gfCNCPoint5[4835] = {X 411.3483, Y 48.2525, Z -6.3333, A 0.000, B 0.000, C 0.000 }
gfCNCPoint5[4836] = {X 410.5596, Y 48.7481, Z -6.3333, A 0.000, B 0.000, C 0.000 }
gfCNCPoint5[4837] = {X 409.6803, Y 49.0557, Z -6.3333, A 0.000, B 0.000, C 0.000 }
gfCNCPoint5[4838] = {X 408.7547, Y 49.1600, Z -6.3333, A 0.000, B 0.000, C 0.000 }
gfCNCPoint5[4839] = {X 402.3112, Y 49.1600, Z -6.3333, A 0.000, B 0.000, C 0.000 }
gfCNCPoint5[4840] = {X 401.3900, Y 49.0567, Z -6.3333, A 0.000, B 0.000, C 0.000 }
gfCNCPoint5[4841] = {X 400.5146, Y 48.7520, Z -6.3333, A 0.000, B 0.000, C 0.000 }
gfCNCPoint5[4842] = {X 399.7283, Y 48.2610, Z -6.3333, A 0.000, B 0.000, C 0.000 }
gfCNCPoint5[4843] = {X 399.0703, Y 47.6081, Z -6.3333, A 0.000, B 0.000, C 0.000 }
gfCNCPoint5[4844] = {X 398.5732, Y 46.8257, Z -6.3333, A 0.000, B 0.000, C 0.000 }
gfCNCPoint5[4845] = {X 398.2617, Y 45.9526, Z -6.3333, A 0.000, B 0.000, C 0.000 }
gfCNCPoint5[4846] = {X 398.1513, Y 45.0322, Z -6.3333, A 0.000, B 0.000, C 0.000 }
gfCNCPoint5[4847] = {X 398.1516, Y 44.1549, Z -6.3333, A 0.000, B 0.000, C 0.000 }
gfCNCPoint5[4848] = {X 398.2616, Y 43.2570, Z -6.3333, A 0.000, B 0.000, C 0.000 }
gfCNCPoint5[4849] = {X 398.5630, Y 42.4041, Z -6.3333, A 0.000, B 0.000, C 0.000 }
gfCNCPoint5[4850] = {X 399.0417, Y 41.6366, Z -6.3333, A 0.000, B 0.000, C 0.000 }
gfCNCPoint5[4851] = {X 399.6750, Y 40.9907, Z -6.3333, A 0.000, B 0.000, C 0.000 }
gfCNCPoint5[4852] = {X 399.6327, Y 31.5586, Z -6.3333, A 0.000, B 0.000, C 0.000 }
gfCNCPoint5[4853] = {X 393.6589, Y 21.1703, Z -6.3333, A 0.000, B 0.000, C 0.000 }
gfCNCPoint5[4854] = {X 392.7687, Y 19.6558, Z -6.3333, A 0.000, B 0.000, C 0.000 }
gfCNCPoint5[4855] = {X 391.8499, Y 18.1584, Z -6.3333, A 0.000, B 0.000, C 0.000 }
gfCNCPoint5[4856] = {X 391.3454, Y 17.4581, Z -6.3333, A 0.000, B 0.000, C 0.000 }
gfCNCPoint5[4857] = {X 390.7551, Y 16.8285, Z -6.3333, A 0.000, B 0.000, C 0.000 }
gfCNCPoint5[4858] = {X 389.9029, Y 16.3569, Z -6.3333, A 0.000, B 0.000, C 0.000 }
gfCNCPoint5[4859] = {X 389.1837, Y 15.7000, Z -6.3333, A 0.000, B 0.000, C 0.000 }
gfCNCPoint5[4860] = {X 388.6371, Y 14.8939, Z -6.3333, A 0.000, B 0.000, C 0.000 }
gfCNCPoint5[4861] = {X 388.2928, Y 13.9828, Z -6.3333, A 0.000, B 0.000, C 0.000 }
gfCNCPoint5[4862] = {X 388.1698, Y 13.0166, Z -6.3333, A 0.000, B 0.000, C 0.000 }
gfCNCPoint5[4863] = {X 388.1696, Y 12.1868, Z -6.3333, A 0.000, B 0.000, C 0.000 }
gfCNCPoint5[4864] = {X 388.2739, Y 11.2611, Z -6.3333, A 0.000, B 0.000, C 0.000 }
gfCNCPoint5[4865] = {X 388.5816, Y 10.3819, Z -6.3333, A 0.000, B 0.000, C 0.000 }
gfCNCPoint5[4866] = {X 389.0772, Y 9.5931, Z -6.3333, A 0.000, B 0.000, C 0.000 }
gfCNCPoint5[4867] = {X 389.7359, Y 8.9344, Z -6.3333, A 0.000, B 0.000, C 0.000 }
gfCNCPoint5[4868] = {X 390.5247, Y 8.4388, Z -6.3333, A 0.000, B 0.000, C 0.000 }
gfCNCPoint5[4869] = {X 391.4039, Y 8.1311, Z -6.3333, A 0.000, B 0.000, C 0.000 }
gfCNCPoint5[4870] = {X 392.3296, Y 8.0268, Z -6.3333, A 0.000, B 0.000, C 0.000 }
gfCNCPoint5[4871] = {X 399.1118, Y 8.0268, Z -6.3333, A 0.000, B 0.000, C 0.000 }
gfCNCPoint5[4872] = {X 400.0374, Y 8.1311, Z -6.3333, A 0.000, B 0.000, C 0.000 }
gfCNCPoint5[4873] = {X 400.9167, Y 8.4388, Z -6.3333, A 0.000, B 0.000, C 0.000 }
gfCNCPoint5[4874] = {X 401.7055, Y 8.9344, Z -6.3333, A 0.000, B 0.000, C 0.000 }
gfCNCPoint5[4875] = {X 402.3642, Y 9.5931, Z -6.3333, A 0.000, B 0.000, C 0.000 }
gfCNCPoint5[4876] = {X 402.8598, Y 10.3819, Z -6.3333, A 0.000, B 0.000, C 0.000 }
gfCNCPoint5[4877] = {X 403.1675, Y 11.2611, Z -6.3333, A 0.000, B 0.000, C 0.000 }
gfCNCPoint5[4878] = {X 403.2718, Y 12.1868, Z -6.3333, A 0.000, B 0.000, C 0.000 }
gfCNCPoint5[4879] = {X 403.2718, Y 12.9782, Z -6.3333, A 0.000, B 0.000, C 0.000 }
gfCNCPoint5[4880] = {X 403.1639, Y 13.9192, Z -6.3333, A 0.000, B 0.000, C 0.000 }
gfCNCPoint5[4881] = {X 402.8459, Y 14.8115, Z -6.3333, A 0.000, B 0.000, C 0.000 }
gfCNCPoint5[4882] = {X 405.3514, Y 19.1340, Z -6.3333, A 0.000, B 0.000, C 0.000 }
gfCNCPoint5[4883] = {X 408.0546, Y 14.7644, Z -6.3333, A 0.000, B 0.000, C 0.000 }
gfCNCPoint5[4884] = {X 407.7575, Y 13.9111, Z -6.3333, A 0.000, B 0.000, C 0.000 }
gfCNCPoint5[4885] = {X 407.6517, Y 13.0137, Z -6.3333, A 0.000, B 0.000, C 0.000 }
gfCNCPoint5[4886] = {X 407.6515, Y 12.1868, Z -6.3333, A 0.000, B 0.000, C 0.000 }
gfCNCPoint5[4887] = {X 407.7558, Y 11.2611, Z -6.3333, A 0.000, B 0.000, C 0.000 }
gfCNCPoint5[4888] = {X 408.0635, Y 10.3819, Z -6.3333, A 0.000, B 0.000, C 0.000 }
gfCNCPoint5[4889] = {X 408.5591, Y 9.5931, Z -6.3333, A 0.000, B 0.000, C 0.000 }
gfCNCPoint5[4890] = {X 409.2178, Y 8.9344, Z -6.3333, A 0.000, B 0.000, C 0.000 }
gfCNCPoint5[4891] = {X 410.0066, Y 8.4388, Z -6.3333, A 0.000, B 0.000, C 0.000 }
gfCNCPoint5[4892] = {X 410.8859, Y 8.1311, Z -6.3333, A 0.000, B 0.000, C 0.000 }
gfCNCPoint5[4893] = {X 411.8115, Y 8.0268, Z -6.3333, A 0.000, B 0.000, C 0.000 }
gfCNCPoint5[4894] = {X 419.3245, Y 8.0268, Z -6.3333, A 0.000, B 0.000, C 0.000 }
gfCNCPoint5[4895] = {X 420.2501, Y 8.1311, Z -6.3333, A 0.000, B 0.000, C 0.000 }
gfCNCPoint5[4896] = {X 421.1294, Y 8.4388, Z -6.3333, A 0.000, B 0.000, C 0.000 }
gfCNCPoint5[4897] = {X 421.9182, Y 8.9344, Z -6.3333, A 0.000, B 0.000, C 0.000 }
gfCNCPoint5[4898] = {X 422.5769, Y 9.5931, Z -6.3333, A 0.000, B 0.000, C 0.000 }
gfCNCPoint5[4899] = {X 423.0725, Y 10.3819, Z -6.3333, A 0.000, B 0.000, C 0.000 }
gfCNCPoint5[4900] = {X 423.3802, Y 11.2611, Z -6.3333, A 0.000, B 0.000, C 0.000 }
gfCNCPoint5[4901] = {X 423.4845, Y 12.1868, Z -6.3333, A 0.000, B 0.000, C 0.000 }
gfCNCPoint5[4902] = {X 423.4845, Y 12.9791, Z -6.3333, A 0.000, B 0.000, C 0.000 }
gfCNCPoint5[4903] = {X 423.3938, Y 13.8210, Z -6.3333, A 0.000, B 0.000, C 0.000 }
gfCNCPoint5[4904] = {X 423.1369, Y 14.6279, Z -6.3333, A 0.000, B 0.000, C 0.000 }
gfCNCPoint5[4905] = {X 422.7241, Y 15.3673, Z -6.3333, A 0.000, B 0.000, C 0.000 }
gfCNCPoint5[4906] = {X 422.1721, Y 16.0094, Z -6.3333, A 0.000, B 0.000, C 0.000 }
gfCNCPoint5[4907] = {X 421.5030, Y 16.5285, Z -6.3333, A 0.000, B 0.000, C 0.000 }
gfCNCPoint5[4908] = {X 420.7439, Y 16.9036, Z -6.3333, A 0.000, B 0.000, C 0.000 }
gfCNCPoint5[4909] = {X 420.0063, Y 17.8914, Z -6.3333, A 0.000, B 0.000, C 0.000 }
gfCNCPoint5[4910] = {X 419.3400, Y 18.9286, Z -6.3333, A 0.000, B 0.000, C 0.000 }
gfCNCPoint5[4911] = {X 417.8582, Y 21.3274, Z -6.3333, A 0.000, B 0.000, C 0.000 }
gfCNCPoint5[4912] = {X 416.0154, Y 24.2871, Z -6.3333, A 0.000, B 0.000, C 0.000 }
gfCNCPoint5[4913] = {X 419.4109, Y 26.4014, Z -6.3333, A 0.000, B 0.000, C 0.000 }
gfCNCPoint5[4914] = {X 415.9475, Y 24.2448, Z -6.3333, A 0.000, B 0.000, C 0.000 }
gfCNCPoint5[4915] = {X 411.3076, Y 31.6967, Z -6.3333, A 0.000, B 0.000, C 0.000 }
gfCNCPoint5[4916] = {X 411.3082, Y 41.0089, Z -6.3333, A 0.000, B 0.000, C 0.000 }
gfCNCPoint5[4917] = {X 411.9451, Y 41.6632, Z -6.3333, A 0.000, B 0.000, C 0.000 }
gfCNCPoint5[4918] = {X 412.4256, Y 42.4397, Z -6.3333, A 0.000, B 0.000, C 0.000 }
gfCNCPoint5[4919] = {X 412.7269, Y 43.3017, Z -6.3333, A 0.000, B 0.000, C 0.000 }
gfCNCPoint5[4920] = {X 412.8347, Y 44.2085, Z -6.3333, A 0.000, B 0.000, C 0.000 }
gfCNCPoint5[4921] = {X 412.8347, Y 45.0002, Z -6.3333, A 0.000, B 0.000, C 0.000 }
gfCNCPoint5[4922] = {X 412.7324, Y 45.9080, Z -6.3333, A 0.000, B 0.000, C 0.000 }
gfCNCPoint5[4923] = {X 412.4306, Y 46.7704, Z -6.3333, A 0.000, B 0.000, C 0.000 }
gfCNCPoint5[4924] = {X 411.9445, Y 47.5439, Z -6.3333, A 0.000, B 0.000, C 0.000 }
gfCNCPoint5[4925] = {X 411.2985, Y 48.1899, Z -6.3333, A 0.000, B 0.000, C 0.000 }
gfCNCPoint5[4926] = {X 410.5249, Y 48.6760, Z -6.3333, A 0.000, B 0.000, C 0.000 }
gfCNCPoint5[4927] = {X 409.6625, Y 48.9777, Z -6.3333, A 0.000, B 0.000, C 0.000 }
gfCNCPoint5[4928] = {X 408.7547, Y 49.0800, Z -6.3333, A 0.000, B 0.000, C 0.000 }
gfCNCPoint5[4929] = {X 402.3112, Y 49.0800, Z -6.3333, A 0.000, B 0.000, C 0.000 }
gfCNCPoint5[4930] = {X 401.4077, Y 48.9787, Z -6.3333, A 0.000, B 0.000, C 0.000 }
gfCNCPoint5[4931] = {X 400.5491, Y 48.6799, Z -6.3333, A 0.000, B 0.000, C 0.000 }
gfCNCPoint5[4932] = {X 399.7780, Y 48.1983, Z -6.3333, A 0.000, B 0.000, C 0.000 }
gfCNCPoint5[4933] = {X 399.1326, Y 47.5579, Z -6.3333, A 0.000, B 0.000, C 0.000 }
gfCNCPoint5[4934] = {X 398.6451, Y 46.7906, Z -6.3333, A 0.000, B 0.000, C 0.000 }
gfCNCPoint5[4935] = {X 398.3396, Y 45.9343, Z -6.3333, A 0.000, B 0.000, C 0.000 }
gfCNCPoint5[4936] = {X 398.2313, Y 45.0316, Z -6.3333, A 0.000, B 0.000, C 0.000 }
gfCNCPoint5[4937] = {X 398.2316, Y 44.1559, Z -6.3333, A 0.000, B 0.000, C 0.000 }
gfCNCPoint5[4938] = {X 398.3416, Y 43.2661, Z -6.3333, A 0.000, B 0.000, C 0.000 }
gfCNCPoint5[4939] = {X 398.6434, Y 42.4218, Z -6.3333, A 0.000, B 0.000, C 0.000 }
gfCNCPoint5[4940] = {X 399.1223, Y 41.6638, Z -6.3333, A 0.000, B 0.000, C 0.000 }
gfCNCPoint5[4941] = {X 399.7552, Y 41.0287, Z -6.3333, A 0.000, B 0.000, C 0.000 }
gfCNCPoint5[4942] = {X 399.7126, Y 31.5371, Z -6.3333, A 0.000, B 0.000, C 0.000 }
gfCNCPoint5[4943] = {X 393.7283, Y 21.1304, Z -6.3333, A 0.000, B 0.000, C 0.000 }
gfCNCPoint5[4944] = {X 392.8373, Y 19.6146, Z -6.3333, A 0.000, B 0.000, C 0.000 }
gfCNCPoint5[4945] = {X 391.9177, Y 18.1159, Z -6.3333, A 0.000, B 0.000, C 0.000 }
gfCNCPoint5[4946] = {X 391.4024, Y 17.4015, Z -6.3333, A 0.000, B 0.000, C 0.000 }
gfCNCPoint5[4947] = {X 390.7989, Y 16.7600, Z -6.3333, A 0.000, B 0.000, C 0.000 }
gfCNCPoint5[4948] = {X 389.9591, Y 16.2987, Z -6.3333, A 0.000, B 0.000, C 0.000 }
gfCNCPoint5[4949] = {X 389.2500, Y 15.6543, Z -6.3333, A 0.000, B 0.000, C 0.000 }
gfCNCPoint5[4950] = {X 388.7108, Y 14.8622, Z -6.3333, A 0.000, B 0.000, C 0.000 }
gfCNCPoint5[4951] = {X 388.3711, Y 13.9663, Z -6.3333, A 0.000, B 0.000, C 0.000 }
gfCNCPoint5[4952] = {X 388.2498, Y 13.0158, Z -6.3333, A 0.000, B 0.000, C 0.000 }
gfCNCPoint5[4953] = {X 388.2496, Y 12.1868, Z -6.3333, A 0.000, B 0.000, C 0.000 }
gfCNCPoint5[4954] = {X 388.3519, Y 11.2789, Z -6.3333, A 0.000, B 0.000, C 0.000 }
gfCNCPoint5[4955] = {X 388.6537, Y 10.4166, Z -6.3333, A 0.000, B 0.000, C 0.000 }
gfCNCPoint5[4956] = {X 389.1398, Y 9.6430, Z -6.3333, A 0.000, B 0.000, C 0.000 }
gfCNCPoint5[4957] = {X 389.7858, Y 8.9969, Z -6.3333, A 0.000, B 0.000, C 0.000 }
gfCNCPoint5[4958] = {X 390.5594, Y 8.5109, Z -6.3333, A 0.000, B 0.000, C 0.000 }
gfCNCPoint5[4959] = {X 391.4217, Y 8.2091, Z -6.3333, A 0.000, B 0.000, C 0.000 }
gfCNCPoint5[4960] = {X 392.3296, Y 8.1068, Z -6.3333, A 0.000, B 0.000, C 0.000 }
gfCNCPoint5[4961] = {X 399.1118, Y 8.1068, Z -6.3333, A 0.000, B 0.000, C 0.000 }
gfCNCPoint5[4962] = {X 400.0196, Y 8.2091, Z -6.3333, A 0.000, B 0.000, C 0.000 }
gfCNCPoint5[4963] = {X 400.8820, Y 8.5109, Z -6.3333, A 0.000, B 0.000, C 0.000 }
gfCNCPoint5[4964] = {X 401.6556, Y 8.9969, Z -6.3333, A 0.000, B 0.000, C 0.000 }
gfCNCPoint5[4965] = {X 402.3016, Y 9.6430, Z -6.3333, A 0.000, B 0.000, C 0.000 }
gfCNCPoint5[4966] = {X 402.7877, Y 10.4166, Z -6.3333, A 0.000, B 0.000, C 0.000 }
gfCNCPoint5[4967] = {X 403.0895, Y 11.2789, Z -6.3333, A 0.000, B 0.000, C 0.000 }
gfCNCPoint5[4968] = {X 403.1918, Y 12.1868, Z -6.3333, A 0.000, B 0.000, C 0.000 }
gfCNCPoint5[4969] = {X 403.1918, Y 12.9782, Z -6.3333, A 0.000, B 0.000, C 0.000 }
gfCNCPoint5[4970] = {X 403.0811, Y 13.9219, Z -6.3333, A 0.000, B 0.000, C 0.000 }
gfCNCPoint5[4971] = {X 402.7551, Y 14.8144, Z -6.3333, A 0.000, B 0.000, C 0.000 }
gfCNCPoint5[4972] = {X 405.3492, Y 19.2896, Z -6.3333, A 0.000, B 0.000, C 0.000 }
gfCNCPoint5[4973] = {X 408.1457, Y 14.7691, Z -6.3333, A 0.000, B 0.000, C 0.000 }
gfCNCPoint5[4974] = {X 408.1090, Y 14.6919, Z -6.3333, A 0.000, B 0.000, C 0.000 }
gfCNCPoint5[4975] = {X 408.0738, Y 14.6138, Z -6.3333, A 0.000, B 0.000, C 0.000 }
gfCNCPoint5[4976] = {X 407.8217, Y 13.8308, Z -6.3333, A 0.000, B 0.000, C 0.000 }
gfCNCPoint5[4977] = {X 407.7317, Y 13.0131, Z -6.3333, A 0.000, B 0.000, C 0.000 }
gfCNCPoint5[4978] = {X 407.7315, Y 12.1868, Z -6.3333, A 0.000, B 0.000, C 0.000 }
gfCNCPoint5[4979] = {X 407.8338, Y 11.2789, Z -6.3333, A 0.000, B 0.000, C 0.000 }
gfCNCPoint5[4980] = {X 408.1356, Y 10.4166, Z -6.3333, A 0.000, B 0.000, C 0.000 }
gfCNCPoint5[4981] = {X 408.6217, Y 9.6430, Z -6.3333, A 0.000, B 0.000, C 0.000 }
gfCNCPoint5[4982] = {X 409.2677, Y 8.9969, Z -6.3333, A 0.000, B 0.000, C 0.000 }
gfCNCPoint5[4983] = {X 410.0413, Y 8.5109, Z -6.3333, A 0.000, B 0.000, C 0.000 }
gfCNCPoint5[4984] = {X 410.9037, Y 8.2091, Z -6.3333, A 0.000, B 0.000, C 0.000 }
gfCNCPoint5[4985] = {X 411.8115, Y 8.1068, Z -6.3333, A 0.000, B 0.000, C 0.000 }
gfCNCPoint5[4986] = {X 419.3245, Y 8.1068, Z -6.3333, A 0.000, B 0.000, C 0.000 }
gfCNCPoint5[4987] = {X 420.2323, Y 8.2091, Z -6.3333, A 0.000, B 0.000, C 0.000 }
gfCNCPoint5[4988] = {X 421.0947, Y 8.5109, Z -6.3333, A 0.000, B 0.000, C 0.000 }
gfCNCPoint5[4989] = {X 421.8683, Y 8.9969, Z -6.3333, A 0.000, B 0.000, C 0.000 }
gfCNCPoint5[4990] = {X 422.5143, Y 9.6430, Z -6.3333, A 0.000, B 0.000, C 0.000 }
gfCNCPoint5[4991] = {X 423.0004, Y 10.4166, Z -6.3333, A 0.000, B 0.000, C 0.000 }
gfCNCPoint5[4992] = {X 423.3022, Y 11.2789, Z -6.3333, A 0.000, B 0.000, C 0.000 }
gfCNCPoint5[4993] = {X 423.4045, Y 12.1868, Z -6.3333, A 0.000, B 0.000, C 0.000 }
gfCNCPoint5[4994] = {X 423.4045, Y 12.9785, Z -6.3333, A 0.000, B 0.000, C 0.000 }
gfCNCPoint5[4995] = {X 423.3147, Y 13.8081, Z -6.3333, A 0.000, B 0.000, C 0.000 }
gfCNCPoint5[4996] = {X 423.0606, Y 14.6028, Z -6.3333, A 0.000, B 0.000, C 0.000 }
gfCNCPoint5[4997] = {X 422.6523, Y 15.3304, Z -6.3333, A 0.000, B 0.000, C 0.000 }
gfCNCPoint5[4998] = {X 422.1064, Y 15.9614, Z -6.3333, A 0.000, B 0.000, C 0.000 }
gfCNCPoint5[4999] = {X 421.4452, Y 16.4703, Z -6.3333, A 0.000, B 0.000, C 0.000 }
gfCNCPoint5[5000] = {X 420.6953, Y 16.8362, Z -6.3333, A 0.000, B 0.000, C 0.000 }
gfCNCPoint5[5001] = {X 419.9471, Y 17.8364, Z -6.3333, A 0.000, B 0.000, C 0.000 }
gfCNCPoint5[5002] = {X 419.2716, Y 18.8871, Z -6.3333, A 0.000, B 0.000, C 0.000 }
gfCNCPoint5[5003] = {X 417.7903, Y 21.2852, Z -6.3333, A 0.000, B 0.000, C 0.000 }
gfCNCPoint5[5004] = {X 415.9475, Y 24.2448, Z -6.3333, A 0.000, B 0.000, C 0.000 }
gfCNCPoint5[5005] = {X 419.3430, Y 26.3591, Z -6.3333, A 0.000, B 0.000, C 0.000 }
gfCNCPoint5[5006] = {X 415.8795, Y 24.2025, Z -6.3333, A 0.000, B 0.000, C 0.000 }
gfCNCPoint5[5007] = {X 411.2276, Y 31.6738, Z -6.3333, A 0.000, B 0.000, C 0.000 }
gfCNCPoint5[5008] = {X 411.2282, Y 41.0468, Z -6.3333, A 0.000, B 0.000, C 0.000 }
gfCNCPoint5[5009] = {X 411.8646, Y 41.6902, Z -6.3333, A 0.000, B 0.000, C 0.000 }
gfCNCPoint5[5010] = {X 412.3452, Y 42.4571, Z -6.3333, A 0.000, B 0.000, C 0.000 }
gfCNCPoint5[5011] = {X 412.6467, Y 43.3103, Z -6.3333, A 0.000, B 0.000, C 0.000 }
gfCNCPoint5[5012] = {X 412.7547, Y 44.2089, Z -6.3333, A 0.000, B 0.000, C 0.000 }
gfCNCPoint5[5013] = {X 412.7545, Y 45.0384, Z -6.3333, A 0.000, B 0.000, C 0.000 }
gfCNCPoint5[5014] = {X 412.6469, Y 45.9222, Z -6.3333, A 0.000, B 0.000, C 0.000 }
gfCNCPoint5[5015] = {X 412.3466, Y 46.7602, Z -6.3333, A 0.000, B 0.000, C 0.000 }
gfCNCPoint5[5016] = {X 411.8683, Y 47.5111, Z -6.3333, A 0.000, B 0.000, C 0.000 }
gfCNCPoint5[5017] = {X 411.2357, Y 48.1376, Z -6.3333, A 0.000, B 0.000, C 0.000 }
gfCNCPoint5[5018] = {X 410.4803, Y 48.6086, Z -6.3333, A 0.000, B 0.000, C 0.000 }
gfCNCPoint5[5019] = {X 409.6394, Y 48.9009, Z -6.3333, A 0.000, B 0.000, C 0.000 }
gfCNCPoint5[5020] = {X 408.7547, Y 49.0000, Z -6.3333, A 0.000, B 0.000, C 0.000 }
gfCNCPoint5[5021] = {X 402.3112, Y 49.0000, Z -6.3333, A 0.000, B 0.000, C 0.000 }
gfCNCPoint5[5022] = {X 401.4211, Y 48.8997, Z -6.3333, A 0.000, B 0.000, C 0.000 }
gfCNCPoint5[5023] = {X 400.5757, Y 48.6039, Z -6.3333, A 0.000, B 0.000, C 0.000 }
gfCNCPoint5[5024] = {X 399.8172, Y 48.1273, Z -6.3333, A 0.000, B 0.000, C 0.000 }
gfCNCPoint5[5025] = {X 399.1839, Y 47.4939, Z -6.3333, A 0.000, B 0.000, C 0.000 }
gfCNCPoint5[5026] = {X 398.7073, Y 46.7355, Z -6.3333, A 0.000, B 0.000, C 0.000 }
gfCNCPoint5[5027] = {X 398.4115, Y 45.8901, Z -6.3333, A 0.000, B 0.000, C 0.000 }
gfCNCPoint5[5028] = {X 398.3112, Y 45.0000, Z -6.3333, A 0.000, B 0.000, C 0.000 }
gfCNCPoint5[5029] = {X 398.3115, Y 44.1569, Z -6.3333, A 0.000, B 0.000, C 0.000 }
gfCNCPoint5[5030] = {X 398.4217, Y 43.2753, Z -6.3333, A 0.000, B 0.000, C 0.000 }
gfCNCPoint5[5031] = {X 398.7237, Y 42.4397, Z -6.3333, A 0.000, B 0.000, C 0.000 }
gfCNCPoint5[5032] = {X 399.2028, Y 41.6913, Z -6.3333, A 0.000, B 0.000, C 0.000 }
gfCNCPoint5[5033] = {X 399.8352, Y 41.0672, Z -6.3333, A 0.000, B 0.000, C 0.000 }
gfCNCPoint5[5034] = {X 399.8367, Y 31.5924, Z -6.3333, A 0.000, B 0.000, C 0.000 }
gfCNCPoint5[5035] = {X 393.7976, Y 21.0906, Z -6.3333, A 0.000, B 0.000, C 0.000 }
gfCNCPoint5[5036] = {X 392.9059, Y 19.5734, Z -6.3333, A 0.000, B 0.000, C 0.000 }
gfCNCPoint5[5037] = {X 391.9855, Y 18.0734, Z -6.3333, A 0.000, B 0.000, C 0.000 }
gfCNCPoint5[5038] = {X 391.4594, Y 17.3449, Z -6.3333, A 0.000, B 0.000, C 0.000 }
gfCNCPoint5[5039] = {X 390.8426, Y 16.6913, Z -6.3333, A 0.000, B 0.000, C 0.000 }
gfCNCPoint5[5040] = {X 390.0091, Y 16.2361, Z -6.3333, A 0.000, B 0.000, C 0.000 }
gfCNCPoint5[5041] = {X 389.3064, Y 15.5972, Z -6.3333, A 0.000, B 0.000, C 0.000 }
gfCNCPoint5[5042] = {X 388.7742, Y 14.8107, Z -6.3333, A 0.000, B 0.000, C 0.000 }
gfCNCPoint5[5043] = {X 388.4423, Y 13.9209, Z -6.3333, A 0.000, B 0.000, C 0.000 }
gfCNCPoint5[5044] = {X 388.3296, Y 12.9780, Z -6.3333, A 0.000, B 0.000, C 0.000 }
gfCNCPoint5[5045] = {X 388.3296, Y 12.1868, Z -6.3333, A 0.000, B 0.000, C 0.000 }
gfCNCPoint5[5046] = {X 388.4299, Y 11.2967, Z -6.3333, A 0.000, B 0.000, C 0.000 }
gfCNCPoint5[5047] = {X 388.7258, Y 10.4513, Z -6.3333, A 0.000, B 0.000, C 0.000 }
gfCNCPoint5[5048] = {X 389.2023, Y 9.6929, Z -6.3333, A 0.000, B 0.000, C 0.000 }
gfCNCPoint5[5049] = {X 389.8357, Y 9.0595, Z -6.3333, A 0.000, B 0.000, C 0.000 }
gfCNCPoint5[5050] = {X 390.5941, Y 8.5829, Z -6.3333, A 0.000, B 0.000, C 0.000 }
gfCNCPoint5[5051] = {X 391.4395, Y 8.2871, Z -6.3333, A 0.000, B 0.000, C 0.000 }
gfCNCPoint5[5052] = {X 392.3296, Y 8.1868, Z -6.3333, A 0.000, B 0.000, C 0.000 }
gfCNCPoint5[5053] = {X 399.1118, Y 8.1868, Z -6.3333, A 0.000, B 0.000, C 0.000 }
gfCNCPoint5[5054] = {X 400.0018, Y 8.2871, Z -6.3333, A 0.000, B 0.000, C 0.000 }
gfCNCPoint5[5055] = {X 400.8473, Y 8.5829, Z -6.3333, A 0.000, B 0.000, C 0.000 }
gfCNCPoint5[5056] = {X 401.6057, Y 9.0595, Z -6.3333, A 0.000, B 0.000, C 0.000 }
gfCNCPoint5[5057] = {X 402.2391, Y 9.6929, Z -6.3333, A 0.000, B 0.000, C 0.000 }
gfCNCPoint5[5058] = {X 402.7156, Y 10.4513, Z -6.3333, A 0.000, B 0.000, C 0.000 }
gfCNCPoint5[5059] = {X 403.0115, Y 11.2967, Z -6.3333, A 0.000, B 0.000, C 0.000 }
gfCNCPoint5[5060] = {X 403.1118, Y 12.1868, Z -6.3333, A 0.000, B 0.000, C 0.000 }
gfCNCPoint5[5061] = {X 403.1115, Y 13.0192, Z -6.3333, A 0.000, B 0.000, C 0.000 }
gfCNCPoint5[5062] = {X 402.9933, Y 13.9442, Z -6.3333, A 0.000, B 0.000, C 0.000 }
gfCNCPoint5[5063] = {X 402.6641, Y 14.8167, Z -6.3333, A 0.000, B 0.000, C 0.000 }
gfCNCPoint5[5064] = {X 405.2576, Y 19.3199, Z -6.3333, A 0.000, B 0.000, C 0.000 }
gfCNCPoint5[5065] = {X 405.3705, Y 19.4073, Z -6.3333, A 0.000, B 0.000, C 0.000 }
gfCNCPoint5[5066] = {X 408.1939, Y 14.8342, Z -6.3333, A 0.000, B 0.000, C 0.000 }
gfCNCPoint5[5067] = {X 408.2428, Y 14.7847, Z -6.3333, A 0.000, B 0.000, C 0.000 }
gfCNCPoint5[5068] = {X 408.1935, Y 14.6839, Z -6.3333, A 0.000, B 0.000, C 0.000 }
gfCNCPoint5[5069] = {X 408.1471, Y 14.5818, Z -6.3333, A 0.000, B 0.000, C 0.000 }
gfCNCPoint5[5070] = {X 407.8963, Y 13.7972, Z -6.3333, A 0.000, B 0.000, C 0.000 }
gfCNCPoint5[5071] = {X 407.8115, Y 12.9780, Z -6.3333, A 0.000, B 0.000, C 0.000 }
gfCNCPoint5[5072] = {X 407.8115, Y 12.1868, Z -6.3333, A 0.000, B 0.000, C 0.000 }
gfCNCPoint5[5073] = {X 407.9118, Y 11.2967, Z -6.3333, A 0.000, B 0.000, C 0.000 }
gfCNCPoint5[5074] = {X 408.2077, Y 10.4513, Z -6.3333, A 0.000, B 0.000, C 0.000 }
gfCNCPoint5[5075] = {X 408.6842, Y 9.6929, Z -6.3333, A 0.000, B 0.000, C 0.000 }
gfCNCPoint5[5076] = {X 409.3176, Y 9.0595, Z -6.3333, A 0.000, B 0.000, C 0.000 }
gfCNCPoint5[5077] = {X 410.0760, Y 8.5829, Z -6.3333, A 0.000, B 0.000, C 0.000 }
gfCNCPoint5[5078] = {X 410.9215, Y 8.2871, Z -6.3333, A 0.000, B 0.000, C 0.000 }
gfCNCPoint5[5079] = {X 411.8115, Y 8.1868, Z -6.3333, A 0.000, B 0.000, C 0.000 }
gfCNCPoint5[5080] = {X 419.3245, Y 8.1868, Z -6.3333, A 0.000, B 0.000, C 0.000 }
gfCNCPoint5[5081] = {X 420.2145, Y 8.2871, Z -6.3333, A 0.000, B 0.000, C 0.000 }
gfCNCPoint5[5082] = {X 421.0600, Y 8.5829, Z -6.3333, A 0.000, B 0.000, C 0.000 }
gfCNCPoint5[5083] = {X 421.8184, Y 9.0595, Z -6.3333, A 0.000, B 0.000, C 0.000 }
gfCNCPoint5[5084] = {X 422.4518, Y 9.6929, Z -6.3333, A 0.000, B 0.000, C 0.000 }
gfCNCPoint5[5085] = {X 422.9283, Y 10.4513, Z -6.3333, A 0.000, B 0.000, C 0.000 }
gfCNCPoint5[5086] = {X 423.2242, Y 11.2967, Z -6.3333, A 0.000, B 0.000, C 0.000 }
gfCNCPoint5[5087] = {X 423.3245, Y 12.1868, Z -6.3333, A 0.000, B 0.000, C 0.000 }
gfCNCPoint5[5088] = {X 423.3245, Y 12.9780, Z -6.3333, A 0.000, B 0.000, C 0.000 }
gfCNCPoint5[5089] = {X 423.2357, Y 13.7951, Z -6.3333, A 0.000, B 0.000, C 0.000 }
gfCNCPoint5[5090] = {X 422.9843, Y 14.5776, Z -6.3333, A 0.000, B 0.000, C 0.000 }
gfCNCPoint5[5091] = {X 422.5805, Y 15.2934, Z -6.3333, A 0.000, B 0.000, C 0.000 }
gfCNCPoint5[5092] = {X 422.0408, Y 15.9133, Z -6.3333, A 0.000, B 0.000, C 0.000 }
gfCNCPoint5[5093] = {X 421.3874, Y 16.4119, Z -6.3333, A 0.000, B 0.000, C 0.000 }
gfCNCPoint5[5094] = {X 420.6470, Y 16.7687, Z -6.3333, A 0.000, B 0.000, C 0.000 }
gfCNCPoint5[5095] = {X 419.8879, Y 17.7814, Z -6.3333, A 0.000, B 0.000, C 0.000 }
gfCNCPoint5[5096] = {X 419.2032, Y 18.8457, Z -6.3333, A 0.000, B 0.000, C 0.000 }
gfCNCPoint5[5097] = {X 417.7223, Y 21.2430, Z -6.3333, A 0.000, B 0.000, C 0.000 }
gfCNCPoint5[5098] = {X 415.8795, Y 24.2025, Z -6.3333, A 0.000, B 0.000, C 0.000 }
gfCNCPoint5[5099] = {X 419.3430, Y 26.3591, Z -6.3333, A 0.000, B 0.000, C 0.000 }
gfCNCPoint5[5100] = {X 419.3430, Y 26.3591, Z -3.3333, A 0.000, B 0.000, C 0.000 }
gfCNCPoint5[5101] = {X 419.3430, Y 26.3591, Z 11.0000, A 0.000, B 0.000, C 0.000 }
gfCNCPoint5[5102] = {X 352.3460, Y -3.5307, Z 11.0000, A 0.000, B 0.000, C 0.000 }
gfCNCPoint5[5103] = {X 352.3460, Y -3.5307, Z -3.3333, A 0.000, B 0.000, C 0.000 }
gfCNCPoint5[5104] = {X 352.3460, Y -3.5307, Z -6.3333, A 0.000, B 0.000, C 0.000 }
gfCNCPoint5[5105] = {X 351.5945, Y 0.4795, Z -6.3333, A 0.000, B 0.000, C 0.000 }
gfCNCPoint5[5106] = {X 351.8708, Y 0.5313, Z -6.3333, A 0.000, B 0.000, C 0.000 }
gfCNCPoint5[5107] = {X 353.8214, Y 1.0218, Z -6.3333, A 0.000, B 0.000, C 0.000 }
gfCNCPoint5[5108] = {X 355.7161, Y 1.6965, Z -6.3333, A 0.000, B 0.000, C 0.000 }
gfCNCPoint5[5109] = {X 357.5377, Y 2.5493, Z -6.3333, A 0.000, B 0.000, C 0.000 }
gfCNCPoint5[5110] = {X 359.2694, Y 3.5724, Z -6.3333, A 0.000, B 0.000, C 0.000 }
gfCNCPoint5[5111] = {X 360.8953, Y 4.7563, Z -6.3333, A 0.000, B 0.000, C 0.000 }
gfCNCPoint5[5112] = {X 362.4006, Y 6.0902, Z -6.3333, A 0.000, B 0.000, C 0.000 }
gfCNCPoint5[5113] = {X 363.7715, Y 7.5620, Z -6.3333, A 0.000, B 0.000, C 0.000 }
gfCNCPoint5[5114] = {X 365.1227, Y 9.3183, Z -6.3333, A 0.000, B 0.000, C 0.000 }
gfCNCPoint5[5115] = {X 366.3137, Y 11.1869, Z -6.3333, A 0.000, B 0.000, C 0.000 }
gfCNCPoint5[5116] = {X 367.3352, Y 13.1533, Z -6.3333, A 0.000, B 0.000, C 0.000 }
gfCNCPoint5[5117] = {X 368.1794, Y 15.2022, Z -6.3333, A 0.000, B 0.000, C 0.000 }
gfCNCPoint5[5118] = {X 368.8395, Y 17.3175, Z -6.3333, A 0.000, B 0.000, C 0.000 }
gfCNCPoint5[5119] = {X 369.3106, Y 19.4827, Z -6.3333, A 0.000, B 0.000, C 0.000 }
gfCNCPoint5[5120] = {X 369.6416, Y 21.8511, Z -6.3333, A 0.000, B 0.000, C 0.000 }
gfCNCPoint5[5121] = {X 369.7933, Y 24.2377, Z -6.3333, A 0.000, B 0.000, C 0.000 }
gfCNCPoint5[5122] = {X 369.7650, Y 26.6289, Z -6.3333, A 0.000, B 0.000, C 0.000 }
gfCNCPoint5[5123] = {X 369.5567, Y 29.0112, Z -6.3333, A 0.000, B 0.000, C 0.000 }
gfCNCPoint5[5124] = {X 369.1697, Y 31.3710, Z -6.3333, A 0.000, B 0.000, C 0.000 }
gfCNCPoint5[5125] = {X 368.6457, Y 33.4753, Z -6.3333, A 0.000, B 0.000, C 0.000 }
gfCNCPoint5[5126] = {X 367.9378, Y 35.5251, Z -6.3333, A 0.000, B 0.000, C 0.000 }
gfCNCPoint5[5127] = {X 367.0518, Y 37.5043, Z -6.3333, A 0.000, B 0.000, C 0.000 }
gfCNCPoint5[5128] = {X 365.9944, Y 39.3976, Z -6.3333, A 0.000, B 0.000, C 0.000 }
gfCNCPoint5[5129] = {X 364.7739, Y 41.1901, Z -6.3333, A 0.000, B 0.000, C 0.000 }
gfCNCPoint5[5130] = {X 364.6580, Y 41.3487, Z -6.3333, A 0.000, B 0.000, C 0.000 }
gfCNCPoint5[5131] = {X 363.2575, Y 43.0257, Z -6.3333, A 0.000, B 0.000, C 0.000 }
gfCNCPoint5[5132] = {X 361.6976, Y 44.5554, Z -6.3333, A 0.000, B 0.000, C 0.000 }
gfCNCPoint5[5133] = {X 359.9935, Y 45.9227, Z -6.3333, A 0.000, B 0.000, C 0.000 }
gfCNCPoint5[5134] = {X 358.1622, Y 47.1141, Z -6.3333, A 0.000, B 0.000, C 0.000 }
gfCNCPoint5[5135] = {X 356.2216, Y 48.1178, Z -6.3333, A 0.000, B 0.000, C 0.000 }
gfCNCPoint5[5136] = {X 354.0239, Y 48.9381, Z -6.3333, A 0.000, B 0.000, C 0.000 }
gfCNCPoint5[5137] = {X 351.7542, Y 49.5305, Z -6.3333, A 0.000, B 0.000, C 0.000 }
gfCNCPoint5[5138] = {X 349.4359, Y 49.8889, Z -6.3333, A 0.000, B 0.000, C 0.000 }
gfCNCPoint5[5139] = {X 347.0933, Y 50.0096, Z -6.3333, A 0.000, B 0.000, C 0.000 }
gfCNCPoint5[5140] = {X 345.0267, Y 49.9747, Z -6.3333, A 0.000, B 0.000, C 0.000 }
gfCNCPoint5[5141] = {X 342.9709, Y 49.7607, Z -6.3333, A 0.000, B 0.000, C 0.000 }
gfCNCPoint5[5142] = {X 340.9414, Y 49.3693, Z -6.3333, A 0.000, B 0.000, C 0.000 }
gfCNCPoint5[5143] = {X 338.9535, Y 48.8033, Z -6.3333, A 0.000, B 0.000, C 0.000 }
gfCNCPoint5[5144] = {X 337.0222, Y 48.0670, Z -6.3333, A 0.000, B 0.000, C 0.000 }
gfCNCPoint5[5145] = {X 335.1620, Y 47.1660, Z -6.3333, A 0.000, B 0.000, C 0.000 }
gfCNCPoint5[5146] = {X 333.5782, Y 46.1877, Z -6.3333, A 0.000, B 0.000, C 0.000 }
gfCNCPoint5[5147] = {X 332.0753, Y 45.0892, Z -6.3333, A 0.000, B 0.000, C 0.000 }
gfCNCPoint5[5148] = {X 330.6625, Y 43.8770, Z -6.3333, A 0.000, B 0.000, C 0.000 }
gfCNCPoint5[5149] = {X 329.7214, Y 43.8765, Z -6.3333, A 0.000, B 0.000, C 0.000 }
gfCNCPoint5[5150] = {X 328.8027, Y 43.6722, Z -6.3333, A 0.000, B 0.000, C 0.000 }
gfCNCPoint5[5151] = {X 327.9501, Y 43.2738, Z -6.3333, A 0.000, B 0.000, C 0.000 }
gfCNCPoint5[5152] = {X 327.2040, Y 42.7002, Z -6.3333, A 0.000, B 0.000, C 0.000 }
gfCNCPoint5[5153] = {X 326.5808, Y 42.0925, Z -6.3333, A 0.000, B 0.000, C 0.000 }
gfCNCPoint5[5154] = {X 325.9523, Y 41.3190, Z -6.3333, A 0.000, B 0.000, C 0.000 }
gfCNCPoint5[5155] = {X 325.5179, Y 40.4220, Z -6.3333, A 0.000, B 0.000, C 0.000 }
gfCNCPoint5[5156] = {X 325.3006, Y 39.4493, Z -6.3333, A 0.000, B 0.000, C 0.000 }
gfCNCPoint5[5157] = {X 325.3120, Y 38.4527, Z -6.3333, A 0.000, B 0.000, C 0.000 }
gfCNCPoint5[5158] = {X 325.5514, Y 37.4852, Z -6.3333, A 0.000, B 0.000, C 0.000 }
gfCNCPoint5[5159] = {X 326.0062, Y 36.5984, Z -6.3333, A 0.000, B 0.000, C 0.000 }
gfCNCPoint5[5160] = {X 330.2396, Y 30.2687, Z -6.3333, A 0.000, B 0.000, C 0.000 }
gfCNCPoint5[5161] = {X 330.8409, Y 29.5518, Z -6.3333, A 0.000, B 0.000, C 0.000 }
gfCNCPoint5[5162] = {X 331.5826, Y 28.9812, Z -6.3333, A 0.000, B 0.000, C 0.000 }
gfCNCPoint5[5163] = {X 332.4297, Y 28.5837, Z -6.3333, A 0.000, B 0.000, C 0.000 }
gfCNCPoint5[5164] = {X 333.3425, Y 28.3780, Z -6.3333, A 0.000, B 0.000, C 0.000 }
gfCNCPoint5[5165] = {X 334.2782, Y 28.3736, Z -6.3333, A 0.000, B 0.000, C 0.000 }
gfCNCPoint5[5166] = {X 335.1929, Y 28.5708, Z -6.3333, A 0.000, B 0.000, C 0.000 }
gfCNCPoint5[5167] = {X 336.0437, Y 28.9604, Z -6.3333, A 0.000, B 0.000, C 0.000 }
gfCNCPoint5[5168] = {X 336.7907, Y 29.5240, Z -6.3333, A 0.000, B 0.000, C 0.000 }
gfCNCPoint5[5169] = {X 337.4284, Y 30.1382, Z -6.3333, A 0.000, B 0.000, C 0.000 }
gfCNCPoint5[5170] = {X 337.9527, Y 30.7608, Z -6.3333, A 0.000, B 0.000, C 0.000 }
gfCNCPoint5[5171] = {X 338.3509, Y 31.4707, Z -6.3333, A 0.000, B 0.000, C 0.000 }
gfCNCPoint5[5172] = {X 338.6089, Y 32.2427, Z -6.3333, A 0.000, B 0.000, C 0.000 }
gfCNCPoint5[5173] = {X 338.7174, Y 33.0494, Z -6.3333, A 0.000, B 0.000, C 0.000 }
gfCNCPoint5[5174] = {X 338.6728, Y 33.8621, Z -6.3333, A 0.000, B 0.000, C 0.000 }
gfCNCPoint5[5175] = {X 339.3239, Y 34.4488, Z -6.3333, A 0.000, B 0.000, C 0.000 }
gfCNCPoint5[5176] = {X 339.9937, Y 35.0139, Z -6.3333, A 0.000, B 0.000, C 0.000 }
gfCNCPoint5[5177] = {X 341.0874, Y 35.7969, Z -6.3333, A 0.000, B 0.000, C 0.000 }
gfCNCPoint5[5178] = {X 342.2716, Y 36.4348, Z -6.3333, A 0.000, B 0.000, C 0.000 }
gfCNCPoint5[5179] = {X 343.5272, Y 36.9173, Z -6.3333, A 0.000, B 0.000, C 0.000 }
gfCNCPoint5[5180] = {X 344.8339, Y 37.2366, Z -6.3333, A 0.000, B 0.000, C 0.000 }
gfCNCPoint5[5181] = {X 346.1705, Y 37.3875, Z -6.3333, A 0.000, B 0.000, C 0.000 }
gfCNCPoint5[5182] = {X 347.5155, Y 37.3676, Z -6.3333, A 0.000, B 0.000, C 0.000 }
gfCNCPoint5[5183] = {X 348.9565, Y 37.1746, Z -6.3333, A 0.000, B 0.000, C 0.000 }
gfCNCPoint5[5184] = {X 350.3468, Y 36.7493, Z -6.3333, A 0.000, B 0.000, C 0.000 }
gfCNCPoint5[5185] = {X 351.6493, Y 36.1033, Z -6.3333, A 0.000, B 0.000, C 0.000 }
gfCNCPoint5[5186] = {X 352.8291, Y 35.2537, Z -6.3333, A 0.000, B 0.000, C 0.000 }
gfCNCPoint5[5187] = {X 353.9825, Y 34.1330, Z -6.3333, A 0.000, B 0.000, C 0.000 }
gfCNCPoint5[5188] = {X 354.9806, Y 32.8721, Z -6.3333, A 0.000, B 0.000, C 0.000 }
gfCNCPoint5[5189] = {X 355.8066, Y 31.4923, Z -6.3333, A 0.000, B 0.000, C 0.000 }
gfCNCPoint5[5190] = {X 356.4465, Y 30.0170, Z -6.3333, A 0.000, B 0.000, C 0.000 }
gfCNCPoint5[5191] = {X 356.8895, Y 28.4711, Z -6.3333, A 0.000, B 0.000, C 0.000 }
gfCNCPoint5[5192] = {X 357.1627, Y 26.7828, Z -6.3333, A 0.000, B 0.000, C 0.000 }
gfCNCPoint5[5193] = {X 357.2740, Y 25.0763, Z -6.3333, A 0.000, B 0.000, C 0.000 }
gfCNCPoint5[5194] = {X 357.2223, Y 23.3669, Z -6.3333, A 0.000, B 0.000, C 0.000 }
gfCNCPoint5[5195] = {X 357.0082, Y 21.6701, Z -6.3333, A 0.000, B 0.000, C 0.000 }
gfCNCPoint5[5196] = {X 356.6545, Y 20.1542, Z -6.3333, A 0.000, B 0.000, C 0.000 }
gfCNCPoint5[5197] = {X 356.1049, Y 18.6979, Z -6.3333, A 0.000, B 0.000, C 0.000 }
gfCNCPoint5[5198] = {X 355.3689, Y 17.3262, Z -6.3333, A 0.000, B 0.000, C 0.000 }
gfCNCPoint5[5199] = {X 354.4594, Y 16.0630, Z -6.3333, A 0.000, B 0.000, C 0.000 }
gfCNCPoint5[5200] = {X 353.5887, Y 15.1360, Z -6.3333, A 0.000, B 0.000, C 0.000 }
gfCNCPoint5[5201] = {X 352.5980, Y 14.3387, Z -6.3333, A 0.000, B 0.000, C 0.000 }
gfCNCPoint5[5202] = {X 351.5062, Y 13.6865, Z -6.3333, A 0.000, B 0.000, C 0.000 }
gfCNCPoint5[5203] = {X 350.3346, Y 13.1920, Z -6.3333, A 0.000, B 0.000, C 0.000 }
gfCNCPoint5[5204] = {X 349.1057, Y 12.8647, Z -6.3333, A 0.000, B 0.000, C 0.000 }
gfCNCPoint5[5205] = {X 347.3454, Y 12.6448, Z -6.3333, A 0.000, B 0.000, C 0.000 }
gfCNCPoint5[5206] = {X 345.5714, Y 12.6601, Z -6.3333, A 0.000, B 0.000, C 0.000 }
gfCNCPoint5[5207] = {X 343.8152, Y 12.9102, Z -6.3333, A 0.000, B 0.000, C 0.000 }
gfCNCPoint5[5208] = {X 342.1075, Y 13.3907, Z -6.3333, A 0.000, B 0.000, C 0.000 }
gfCNCPoint5[5209] = {X 340.4785, Y 14.0933, Z -6.3333, A 0.000, B 0.000, C 0.000 }
gfCNCPoint5[5210] = {X 338.9570, Y 15.0054, Z -6.3333, A 0.000, B 0.000, C 0.000 }
gfCNCPoint5[5211] = {X 338.9180, Y 15.8501, Z -6.3333, A 0.000, B 0.000, C 0.000 }
gfCNCPoint5[5212] = {X 338.7153, Y 16.6711, Z -6.3333, A 0.000, B 0.000, C 0.000 }
gfCNCPoint5[5213] = {X 338.3565, Y 17.4368, Z -6.3333, A 0.000, B 0.000, C 0.000 }
gfCNCPoint5[5214] = {X 337.8554, Y 18.1180, Z -6.3333, A 0.000, B 0.000, C 0.000 }
gfCNCPoint5[5215] = {X 337.2312, Y 18.6885, Z -6.3333, A 0.000, B 0.000, C 0.000 }
gfCNCPoint5[5216] = {X 336.5140, Y 19.2162, Z -6.3333, A 0.000, B 0.000, C 0.000 }
gfCNCPoint5[5217] = {X 335.6982, Y 19.6754, Z -6.3333, A 0.000, B 0.000, C 0.000 }
gfCNCPoint5[5218] = {X 334.8027, Y 19.9480, Z -6.3333, A 0.000, B 0.000, C 0.000 }
gfCNCPoint5[5219] = {X 333.8694, Y 20.0213, Z -6.3333, A 0.000, B 0.000, C 0.000 }
gfCNCPoint5[5220] = {X 332.9422, Y 19.8919, Z -6.3333, A 0.000, B 0.000, C 0.000 }
gfCNCPoint5[5221] = {X 332.0647, Y 19.5657, Z -6.3333, A 0.000, B 0.000, C 0.000 }
gfCNCPoint5[5222] = {X 331.2781, Y 19.0582, Z -6.3333, A 0.000, B 0.000, C 0.000 }
gfCNCPoint5[5223] = {X 330.6193, Y 18.3931, Z -6.3333, A 0.000, B 0.000, C 0.000 }
gfCNCPoint5[5224] = {X 330.1192, Y 17.6017, Z -6.3333, A 0.000, B 0.000, C 0.000 }
gfCNCPoint5[5225] = {X 326.5942, Y 10.3502, Z -6.3333, A 0.000, B 0.000, C 0.000 }
gfCNCPoint5[5226] = {X 326.2930, Y 9.5271, Z -6.3333, A 0.000, B 0.000, C 0.000 }
gfCNCPoint5[5227] = {X 326.1640, Y 8.6602, Z -6.3333, A 0.000, B 0.000, C 0.000 }
gfCNCPoint5[5228] = {X 326.2128, Y 7.7851, Z -6.3333, A 0.000, B 0.000, C 0.000 }
gfCNCPoint5[5229] = {X 326.4371, Y 6.9378, Z -6.3333, A 0.000, B 0.000, C 0.000 }
gfCNCPoint5[5230] = {X 326.8279, Y 6.1532, Z -6.3333, A 0.000, B 0.000, C 0.000 }
gfCNCPoint5[5231] = {X 327.3690, Y 5.4637, Z -6.3333, A 0.000, B 0.000, C 0.000 }
gfCNCPoint5[5232] = {X 328.0381, Y 4.8976, Z -6.3333, A 0.000, B 0.000, C 0.000 }
gfCNCPoint5[5233] = {X 328.7084, Y 4.4386, Z -6.3333, A 0.000, B 0.000, C 0.000 }
gfCNCPoint5[5234] = {X 329.5887, Y 3.9824, Z -6.3333, A 0.000, B 0.000, C 0.000 }
gfCNCPoint5[5235] = {X 330.5499, Y 3.7390, Z -6.3333, A 0.000, B 0.000, C 0.000 }
gfCNCPoint5[5236] = {X 331.5412, Y 3.7211, Z -6.3333, A 0.000, B 0.000, C 0.000 }
gfCNCPoint5[5237] = {X 332.5105, Y 3.9297, Z -6.3333, A 0.000, B 0.000, C 0.000 }
gfCNCPoint5[5238] = {X 334.1673, Y 3.0114, Z -6.3333, A 0.000, B 0.000, C 0.000 }
gfCNCPoint5[5239] = {X 335.8815, Y 2.2051, Z -6.3333, A 0.000, B 0.000, C 0.000 }
gfCNCPoint5[5240] = {X 337.9804, Y 1.3869, Z -6.3333, A 0.000, B 0.000, C 0.000 }
gfCNCPoint5[5241] = {X 340.1416, Y 0.7513, Z -6.3333, A 0.000, B 0.000, C 0.000 }
gfCNCPoint5[5242] = {X 342.3493, Y 0.3030, Z -6.3333, A 0.000, B 0.000, C 0.000 }
gfCNCPoint5[5243] = {X 344.5873, Y 0.0453, Z -6.3333, A 0.000, B 0.000, C 0.000 }
gfCNCPoint5[5244] = {X 346.8391, Y -0.0199, Z -6.3333, A 0.000, B 0.000, C 0.000 }
gfCNCPoint5[5245] = {X 349.0883, Y 0.1079, Z -6.3333, A 0.000, B 0.000, C 0.000 }
gfCNCPoint5[5246] = {X 351.3182, Y 0.4277, Z -6.3333, A 0.000, B 0.000, C 0.000 }
gfCNCPoint5[5247] = {X 351.5945, Y 0.4795, Z -6.3333, A 0.000, B 0.000, C 0.000 }
gfCNCPoint5[5248] = {X 352.3313, Y -3.4520, Z -6.3333, A 0.000, B 0.000, C 0.000 }
gfCNCPoint5[5249] = {X 351.5798, Y 0.5581, Z -6.3333, A 0.000, B 0.000, C 0.000 }
gfCNCPoint5[5250] = {X 351.8555, Y 0.6098, Z -6.3333, A 0.000, B 0.000, C 0.000 }
gfCNCPoint5[5251] = {X 353.7986, Y 1.0985, Z -6.3333, A 0.000, B 0.000, C 0.000 }
gfCNCPoint5[5252] = {X 355.6860, Y 1.7707, Z -6.3333, A 0.000, B 0.000, C 0.000 }
gfCNCPoint5[5253] = {X 357.5006, Y 2.6202, Z -6.3333, A 0.000, B 0.000, C 0.000 }
gfCNCPoint5[5254] = {X 359.2256, Y 3.6394, Z -6.3333, A 0.000, B 0.000, C 0.000 }
gfCNCPoint5[5255] = {X 360.8453, Y 4.8187, Z -6.3333, A 0.000, B 0.000, C 0.000 }
gfCNCPoint5[5256] = {X 362.3448, Y 6.1475, Z -6.3333, A 0.000, B 0.000, C 0.000 }
gfCNCPoint5[5257] = {X 363.7104, Y 7.6136, Z -6.3333, A 0.000, B 0.000, C 0.000 }
gfCNCPoint5[5258] = {X 365.0573, Y 9.3644, Z -6.3333, A 0.000, B 0.000, C 0.000 }
gfCNCPoint5[5259] = {X 366.2445, Y 11.2271, Z -6.3333, A 0.000, B 0.000, C 0.000 }
gfCNCPoint5[5260] = {X 367.2628, Y 13.1873, Z -6.3333, A 0.000, B 0.000, C 0.000 }
gfCNCPoint5[5261] = {X 368.1042, Y 15.2296, Z -6.3333, A 0.000, B 0.000, C 0.000 }
gfCNCPoint5[5262] = {X 368.7623, Y 17.3382, Z -6.3333, A 0.000, B 0.000, C 0.000 }
gfCNCPoint5[5263] = {X 369.2318, Y 19.4966, Z -6.3333, A 0.000, B 0.000, C 0.000 }
gfCNCPoint5[5264] = {X 369.5619, Y 21.8590, Z -6.3333, A 0.000, B 0.000, C 0.000 }
gfCNCPoint5[5265] = {X 369.7133, Y 24.2396, Z -6.3333, A 0.000, B 0.000, C 0.000 }
gfCNCPoint5[5266] = {X 369.6851, Y 26.6248, Z -6.3333, A 0.000, B 0.000, C 0.000 }
gfCNCPoint5[5267] = {X 369.4773, Y 29.0012, Z -6.3333, A 0.000, B 0.000, C 0.000 }
gfCNCPoint5[5268] = {X 369.0913, Y 31.3551, Z -6.3333, A 0.000, B 0.000, C 0.000 }
gfCNCPoint5[5269] = {X 368.5689, Y 33.4526, Z -6.3333, A 0.000, B 0.000, C 0.000 }
gfCNCPoint5[5270] = {X 367.8634, Y 35.4958, Z -6.3333, A 0.000, B 0.000, C 0.000 }
gfCNCPoint5[5271] = {X 366.9801, Y 37.4687, Z -6.3333, A 0.000, B 0.000, C 0.000 }
gfCNCPoint5[5272] = {X 365.9261, Y 39.3559, Z -6.3333, A 0.000, B 0.000, C 0.000 }
gfCNCPoint5[5273] = {X 364.7095, Y 41.1426, Z -6.3333, A 0.000, B 0.000, C 0.000 }
gfCNCPoint5[5274] = {X 364.5937, Y 41.3010, Z -6.3333, A 0.000, B 0.000, C 0.000 }
gfCNCPoint5[5275] = {X 363.1985, Y 42.9717, Z -6.3333, A 0.000, B 0.000, C 0.000 }
gfCNCPoint5[5276] = {X 361.6445, Y 44.4956, Z -6.3333, A 0.000, B 0.000, C 0.000 }
gfCNCPoint5[5277] = {X 359.9468, Y 45.8577, Z -6.3333, A 0.000, B 0.000, C 0.000 }
gfCNCPoint5[5278] = {X 358.1224, Y 47.0447, Z -6.3333, A 0.000, B 0.000, C 0.000 }
gfCNCPoint5[5279] = {X 356.1891, Y 48.0447, Z -6.3333, A 0.000, B 0.000, C 0.000 }
gfCNCPoint5[5280] = {X 353.9990, Y 48.8621, Z -6.3333, A 0.000, B 0.000, C 0.000 }
gfCNCPoint5[5281] = {X 351.7371, Y 49.4524, Z -6.3333, A 0.000, B 0.000, C 0.000 }
gfCNCPoint5[5282] = {X 349.4268, Y 49.8094, Z -6.3333, A 0.000, B 0.000, C 0.000 }
gfCNCPoint5[5283] = {X 347.0922, Y 49.9296, Z -6.3333, A 0.000, B 0.000, C 0.000 }
gfCNCPoint5[5284] = {X 345.0325, Y 49.8949, Z -6.3333, A 0.000, B 0.000, C 0.000 }
gfCNCPoint5[5285] = {X 342.9835, Y 49.6817, Z -6.3333, A 0.000, B 0.000, C 0.000 }
gfCNCPoint5[5286] = {X 340.9608, Y 49.2917, Z -6.3333, A 0.000, B 0.000, C 0.000 }
gfCNCPoint5[5287] = {X 338.9796, Y 48.7276, Z -6.3333, A 0.000, B 0.000, C 0.000 }
gfCNCPoint5[5288] = {X 337.0547, Y 47.9939, Z -6.3333, A 0.000, B 0.000, C 0.000 }
gfCNCPoint5[5289] = {X 335.2007, Y 47.0960, Z -6.3333, A 0.000, B 0.000, C 0.000 }
gfCNCPoint5[5290] = {X 333.6123, Y 46.1142, Z -6.3333, A 0.000, B 0.000, C 0.000 }
gfCNCPoint5[5291] = {X 332.1056, Y 45.0111, Z -6.3333, A 0.000, B 0.000, C 0.000 }
gfCNCPoint5[5292] = {X 330.6900, Y 43.7933, Z -6.3333, A 0.000, B 0.000, C 0.000 }
gfCNCPoint5[5293] = {X 329.7573, Y 43.7998, Z -6.3333, A 0.000, B 0.000, C 0.000 }
gfCNCPoint5[5294] = {X 328.8457, Y 43.6022, Z -6.3333, A 0.000, B 0.000, C 0.000 }
gfCNCPoint5[5295] = {X 327.9995, Y 43.2101, Z -6.3333, A 0.000, B 0.000, C 0.000 }
gfCNCPoint5[5296] = {X 327.2594, Y 42.6425, Z -6.3333, A 0.000, B 0.000, C 0.000 }
gfCNCPoint5[5297] = {X 326.6366, Y 42.0352, Z -6.3333, A 0.000, B 0.000, C 0.000 }
gfCNCPoint5[5298] = {X 326.0198, Y 41.2760, Z -6.3333, A 0.000, B 0.000, C 0.000 }
gfCNCPoint5[5299] = {X 325.5934, Y 40.3956, Z -6.3333, A 0.000, B 0.000, C 0.000 }
gfCNCPoint5[5300] = {X 325.3802, Y 39.4410, Z -6.3333, A 0.000, B 0.000, C 0.000 }
gfCNCPoint5[5301] = {X 325.3913, Y 38.4628, Z -6.3333, A 0.000, B 0.000, C 0.000 }
gfCNCPoint5[5302] = {X 325.6264, Y 37.5133, Z -6.3333, A 0.000, B 0.000, C 0.000 }
gfCNCPoint5[5303] = {X 326.0727, Y 36.6429, Z -6.3333, A 0.000, B 0.000, C 0.000 }
gfCNCPoint5[5304] = {X 330.3061, Y 30.3131, Z -6.3333, A 0.000, B 0.000, C 0.000 }
gfCNCPoint5[5305] = {X 330.8963, Y 29.6095, Z -6.3333, A 0.000, B 0.000, C 0.000 }
gfCNCPoint5[5306] = {X 331.6242, Y 29.0495, Z -6.3333, A 0.000, B 0.000, C 0.000 }
gfCNCPoint5[5307] = {X 332.4556, Y 28.6594, Z -6.3333, A 0.000, B 0.000, C 0.000 }
gfCNCPoint5[5308] = {X 333.3515, Y 28.4575, Z -6.3333, A 0.000, B 0.000, C 0.000 }
gfCNCPoint5[5309] = {X 334.2699, Y 28.4532, Z -6.3333, A 0.000, B 0.000, C 0.000 }
gfCNCPoint5[5310] = {X 335.1677, Y 28.6467, Z -6.3333, A 0.000, B 0.000, C 0.000 }
gfCNCPoint5[5311] = {X 336.0027, Y 29.0291, Z -6.3333, A 0.000, B 0.000, C 0.000 }
gfCNCPoint5[5312] = {X 336.7358, Y 29.5823, Z -6.3333, A 0.000, B 0.000, C 0.000 }
gfCNCPoint5[5313] = {X 337.3723, Y 30.1953, Z -6.3333, A 0.000, B 0.000, C 0.000 }
gfCNCPoint5[5314] = {X 337.8917, Y 30.8133, Z -6.3333, A 0.000, B 0.000, C 0.000 }
gfCNCPoint5[5315] = {X 338.2845, Y 31.5185, Z -6.3333, A 0.000, B 0.000, C 0.000 }
gfCNCPoint5[5316] = {X 338.5366, Y 32.2854, Z -6.3333, A 0.000, B 0.000, C 0.000 }
gfCNCPoint5[5317] = {X 338.6387, Y 33.0861, Z -6.3333, A 0.000, B 0.000, C 0.000 }
gfCNCPoint5[5318] = {X 338.5872, Y 33.8917, Z -6.3333, A 0.000, B 0.000, C 0.000 }
gfCNCPoint5[5319] = {X 339.2553, Y 34.4951, Z -6.3333, A 0.000, B 0.000, C 0.000 }
gfCNCPoint5[5320] = {X 339.9431, Y 35.0758, Z -6.3333, A 0.000, B 0.000, C 0.000 }
gfCNCPoint5[5321] = {X 341.0450, Y 35.8647, Z -6.3333, A 0.000, B 0.000, C 0.000 }
gfCNCPoint5[5322] = {X 342.2379, Y 36.5074, Z -6.3333, A 0.000, B 0.000, C 0.000 }
gfCNCPoint5[5323] = {X 343.5028, Y 36.9935, Z -6.3333, A 0.000, B 0.000, C 0.000 }
gfCNCPoint5[5324] = {X 344.8192, Y 37.3152, Z -6.3333, A 0.000, B 0.000, C 0.000 }
gfCNCPoint5[5325] = {X 346.1657, Y 37.4674, Z -6.3333, A 0.000, B 0.000, C 0.000 }
gfCNCPoint5[5326] = {X 347.5207, Y 37.4474, Z -6.3333, A 0.000, B 0.000, C 0.000 }
gfCNCPoint5[5327] = {X 348.6865, Y 37.3105, Z -6.3333, A 0.000, B 0.000, C 0.000 }
gfCNCPoint5[5328] = {X 349.8245, Y 37.0226, Z -6.3333, A 0.000, B 0.000, C 0.000 }
gfCNCPoint5[5329] = {X 350.9151, Y 36.5886, Z -6.3333, A 0.000, B 0.000, C 0.000 }
gfCNCPoint5[5330] = {X 351.9398, Y 36.0160, Z -6.3333, A 0.000, B 0.000, C 0.000 }
gfCNCPoint5[5331] = {X 352.8810, Y 35.3145, Z -6.3333, A 0.000, B 0.000, C 0.000 }
gfCNCPoint5[5332] = {X 354.0418, Y 34.1866, Z -6.3333, A 0.000, B 0.000, C 0.000 }
gfCNCPoint5[5333] = {X 355.0465, Y 32.9175, Z -6.3333, A 0.000, B 0.000, C 0.000 }
gfCNCPoint5[5334] = {X 355.8778, Y 31.5287, Z -6.3333, A 0.000, B 0.000, C 0.000 }
gfCNCPoint5[5335] = {X 356.5219, Y 30.0438, Z -6.3333, A 0.000, B 0.000, C 0.000 }
gfCNCPoint5[5336] = {X 356.9677, Y 28.4878, Z -6.3333, A 0.000, B 0.000, C 0.000 }
gfCNCPoint5[5337] = {X 357.2422, Y 26.7920, Z -6.3333, A 0.000, B 0.000, C 0.000 }
gfCNCPoint5[5338] = {X 357.3540, Y 25.0778, Z -6.3333, A 0.000, B 0.000, C 0.000 }
gfCNCPoint5[5339] = {X 357.3021, Y 23.3607, Z -6.3333, A 0.000, B 0.000, C 0.000 }
gfCNCPoint5[5340] = {X 357.0870, Y 21.6563, Z -6.3333, A 0.000, B 0.000, C 0.000 }
gfCNCPoint5[5341] = {X 356.7308, Y 20.1304, Z -6.3333, A 0.000, B 0.000, C 0.000 }
gfCNCPoint5[5342] = {X 356.1775, Y 18.6644, Z -6.3333, A 0.000, B 0.000, C 0.000 }
gfCNCPoint5[5343] = {X 355.4367, Y 17.2837, Z -6.3333, A 0.000, B 0.000, C 0.000 }
gfCNCPoint5[5344] = {X 354.5211, Y 16.0120, Z -6.3333, A 0.000, B 0.000, C 0.000 }
gfCNCPoint5[5345] = {X 353.6429, Y 15.0771, Z -6.3333, A 0.000, B 0.000, C 0.000 }
gfCNCPoint5[5346] = {X 352.6435, Y 14.2729, Z -6.3333, A 0.000, B 0.000, C 0.000 }
gfCNCPoint5[5347] = {X 351.5422, Y 13.6151, Z -6.3333, A 0.000, B 0.000, C 0.000 }
gfCNCPoint5[5348] = {X 350.3604, Y 13.1163, Z -6.3333, A 0.000, B 0.000, C 0.000 }
gfCNCPoint5[5349] = {X 349.1209, Y 12.7862, Z -6.3333, A 0.000, B 0.000, C 0.000 }
gfCNCPoint5[5350] = {X 347.3425, Y 12.5645, Z -6.3333, A 0.000, B 0.000, C 0.000 }
gfCNCPoint5[5351] = {X 345.5505, Y 12.5814, Z -6.3333, A 0.000, B 0.000, C 0.000 }
gfCNCPoint5[5352] = {X 343.7767, Y 12.8365, Z -6.3333, A 0.000, B 0.000, C 0.000 }
gfCNCPoint5[5353] = {X 342.0526, Y 13.3253, Z -6.3333, A 0.000, B 0.000, C 0.000 }
gfCNCPoint5[5354] = {X 340.4088, Y 14.0392, Z -6.3333, A 0.000, B 0.000, C 0.000 }
gfCNCPoint5[5355] = {X 338.8746, Y 14.9653, Z -6.3333, A 0.000, B 0.000, C 0.000 }
gfCNCPoint5[5356] = {X 338.8438, Y 15.8035, Z -6.3333, A 0.000, B 0.000, C 0.000 }
gfCNCPoint5[5357] = {X 338.6487, Y 16.6193, Z -6.3333, A 0.000, B 0.000, C 0.000 }
gfCNCPoint5[5358] = {X 338.2967, Y 17.3807, Z -6.3333, A 0.000, B 0.000, C 0.000 }
gfCNCPoint5[5359] = {X 337.8018, Y 18.0579, Z -6.3333, A 0.000, B 0.000, C 0.000 }
gfCNCPoint5[5360] = {X 337.1832, Y 18.6244, Z -6.3333, A 0.000, B 0.000, C 0.000 }
gfCNCPoint5[5361] = {X 336.4675, Y 19.1512, Z -6.3333, A 0.000, B 0.000, C 0.000 }
gfCNCPoint5[5362] = {X 335.6668, Y 19.6018, Z -6.3333, A 0.000, B 0.000, C 0.000 }
gfCNCPoint5[5363] = {X 334.7878, Y 19.8694, Z -6.3333, A 0.000, B 0.000, C 0.000 }
gfCNCPoint5[5364] = {X 333.8718, Y 19.9414, Z -6.3333, A 0.000, B 0.000, C 0.000 }
gfCNCPoint5[5365] = {X 332.9618, Y 19.8143, Z -6.3333, A 0.000, B 0.000, C 0.000 }
gfCNCPoint5[5366] = {X 332.1006, Y 19.4942, Z -6.3333, A 0.000, B 0.000, C 0.000 }
gfCNCPoint5[5367] = {X 331.3285, Y 18.9960, Z -6.3333, A 0.000, B 0.000, C 0.000 }
gfCNCPoint5[5368] = {X 330.6819, Y 18.3433, Z -6.3333, A 0.000, B 0.000, C 0.000 }
gfCNCPoint5[5369] = {X 330.1911, Y 17.5665, Z -6.3333, A 0.000, B 0.000, C 0.000 }
gfCNCPoint5[5370] = {X 326.6662, Y 10.3152, Z -6.3333, A 0.000, B 0.000, C 0.000 }
gfCNCPoint5[5371] = {X 326.3374, Y 9.3676, Z -6.3333, A 0.000, B 0.000, C 0.000 }
gfCNCPoint5[5372] = {X 326.2405, Y 8.3693, Z -6.3333, A 0.000, B 0.000, C 0.000 }
gfCNCPoint5[5373] = {X 326.3807, Y 7.3762, Z -6.3333, A 0.000, B 0.000, C 0.000 }
gfCNCPoint5[5374] = {X 326.7504, Y 6.4438, Z -6.3333, A 0.000, B 0.000, C 0.000 }
gfCNCPoint5[5375] = {X 327.3287, Y 5.6243, Z -6.3333, A 0.000, B 0.000, C 0.000 }
gfCNCPoint5[5376] = {X 328.0833, Y 4.9636, Z -6.3333, A 0.000, B 0.000, C 0.000 }
gfCNCPoint5[5377] = {X 328.7533, Y 4.5047, Z -6.3333, A 0.000, B 0.000, C 0.000 }
gfCNCPoint5[5378] = {X 329.6259, Y 4.0538, Z -6.3333, A 0.000, B 0.000, C 0.000 }
gfCNCPoint5[5379] = {X 330.5789, Y 3.8158, Z -6.3333, A 0.000, B 0.000, C 0.000 }
gfCNCPoint5[5380] = {X 331.5610, Y 3.8035, Z -6.3333, A 0.000, B 0.000, C 0.000 }
gfCNCPoint5[5381] = {X 332.5197, Y 4.0175, Z -6.3333, A 0.000, B 0.000, C 0.000 }
gfCNCPoint5[5382] = {X 334.1874, Y 3.0910, Z -6.3333, A 0.000, B 0.000, C 0.000 }
gfCNCPoint5[5383] = {X 335.9135, Y 2.2785, Z -6.3333, A 0.000, B 0.000, C 0.000 }
gfCNCPoint5[5384] = {X 338.0060, Y 1.4627, Z -6.3333, A 0.000, B 0.000, C 0.000 }
gfCNCPoint5[5385] = {X 340.1607, Y 0.8290, Z -6.3333, A 0.000, B 0.000, C 0.000 }
gfCNCPoint5[5386] = {X 342.3617, Y 0.3820, Z -6.3333, A 0.000, B 0.000, C 0.000 }
gfCNCPoint5[5387] = {X 344.5929, Y 0.1251, Z -6.3333, A 0.000, B 0.000, C 0.000 }
gfCNCPoint5[5388] = {X 346.8379, Y 0.0601, Z -6.3333, A 0.000, B 0.000, C 0.000 }
gfCNCPoint5[5389] = {X 349.0803, Y 0.1875, Z -6.3333, A 0.000, B 0.000, C 0.000 }
gfCNCPoint5[5390] = {X 351.3035, Y 0.5064, Z -6.3333, A 0.000, B 0.000, C 0.000 }
gfCNCPoint5[5391] = {X 351.5798, Y 0.5581, Z -6.3333, A 0.000, B 0.000, C 0.000 }
gfCNCPoint5[5392] = {X 352.3166, Y -3.3734, Z -6.3333, A 0.000, B 0.000, C 0.000 }
gfCNCPoint5[5393] = {X 351.5650, Y 0.6368, Z -6.3333, A 0.000, B 0.000, C 0.000 }
gfCNCPoint5[5394] = {X 351.8403, Y 0.6884, Z -6.3333, A 0.000, B 0.000, C 0.000 }
gfCNCPoint5[5395] = {X 353.7758, Y 1.1752, Z -6.3333, A 0.000, B 0.000, C 0.000 }
gfCNCPoint5[5396] = {X 355.6560, Y 1.8448, Z -6.3333, A 0.000, B 0.000, C 0.000 }
gfCNCPoint5[5397] = {X 357.4635, Y 2.6911, Z -6.3333, A 0.000, B 0.000, C 0.000 }
gfCNCPoint5[5398] = {X 359.1819, Y 3.7063, Z -6.3333, A 0.000, B 0.000, C 0.000 }
gfCNCPoint5[5399] = {X 360.7953, Y 4.8812, Z -6.3333, A 0.000, B 0.000, C 0.000 }
gfCNCPoint5[5400] = {X 362.2890, Y 6.2049, Z -6.3333, A 0.000, B 0.000, C 0.000 }
gfCNCPoint5[5401] = {X 363.6494, Y 7.6653, Z -6.3333, A 0.000, B 0.000, C 0.000 }
gfCNCPoint5[5402] = {X 364.9919, Y 9.4105, Z -6.3333, A 0.000, B 0.000, C 0.000 }
gfCNCPoint5[5403] = {X 366.1753, Y 11.2673, Z -6.3333, A 0.000, B 0.000, C 0.000 }
gfCNCPoint5[5404] = {X 367.1903, Y 13.2212, Z -6.3333, A 0.000, B 0.000, C 0.000 }
gfCNCPoint5[5405] = {X 368.0290, Y 15.2570, Z -6.3333, A 0.000, B 0.000, C 0.000 }
gfCNCPoint5[5406] = {X 368.6850, Y 17.3589, Z -6.3333, A 0.000, B 0.000, C 0.000 }
gfCNCPoint5[5407] = {X 369.1530, Y 19.5104, Z -6.3333, A 0.000, B 0.000, C 0.000 }
gfCNCPoint5[5408] = {X 369.4823, Y 21.8669, Z -6.3333, A 0.000, B 0.000, C 0.000 }
gfCNCPoint5[5409] = {X 369.6333, Y 24.2415, Z -6.3333, A 0.000, B 0.000, C 0.000 }
gfCNCPoint5[5410] = {X 369.6052, Y 26.6208, Z -6.3333, A 0.000, B 0.000, C 0.000 }
gfCNCPoint5[5411] = {X 369.3980, Y 28.9912, Z -6.3333, A 0.000, B 0.000, C 0.000 }
gfCNCPoint5[5412] = {X 369.0129, Y 31.3392, Z -6.3333, A 0.000, B 0.000, C 0.000 }
gfCNCPoint5[5413] = {X 368.4922, Y 33.4300, Z -6.3333, A 0.000, B 0.000, C 0.000 }
gfCNCPoint5[5414] = {X 367.7889, Y 35.4665, Z -6.3333, A 0.000, B 0.000, C 0.000 }
gfCNCPoint5[5415] = {X 366.9085, Y 37.4330, Z -6.3333, A 0.000, B 0.000, C 0.000 }
gfCNCPoint5[5416] = {X 365.8579, Y 39.3141, Z -6.3333, A 0.000, B 0.000, C 0.000 }
gfCNCPoint5[5417] = {X 364.6452, Y 41.0950, Z -6.3333, A 0.000, B 0.000, C 0.000 }
gfCNCPoint5[5418] = {X 364.5295, Y 41.2534, Z -6.3333, A 0.000, B 0.000, C 0.000 }
gfCNCPoint5[5419] = {X 363.1396, Y 42.9176, Z -6.3333, A 0.000, B 0.000, C 0.000 }
gfCNCPoint5[5420] = {X 361.5913, Y 44.4358, Z -6.3333, A 0.000, B 0.000, C 0.000 }
gfCNCPoint5[5421] = {X 359.9001, Y 45.7928, Z -6.3333, A 0.000, B 0.000, C 0.000 }
gfCNCPoint5[5422] = {X 358.0826, Y 46.9753, Z -6.3333, A 0.000, B 0.000, C 0.000 }
gfCNCPoint5[5423] = {X 356.1567, Y 47.9716, Z -6.3333, A 0.000, B 0.000, C 0.000 }
gfCNCPoint5[5424] = {X 353.9741, Y 48.7861, Z -6.3333, A 0.000, B 0.000, C 0.000 }
gfCNCPoint5[5425] = {X 351.7199, Y 49.3742, Z -6.3333, A 0.000, B 0.000, C 0.000 }
gfCNCPoint5[5426] = {X 349.4176, Y 49.7300, Z -6.3333, A 0.000, B 0.000, C 0.000 }
gfCNCPoint5[5427] = {X 347.0911, Y 49.8496, Z -6.3333, A 0.000, B 0.000, C 0.000 }
gfCNCPoint5[5428] = {X 345.0383, Y 49.8151, Z -6.3333, A 0.000, B 0.000, C 0.000 }
gfCNCPoint5[5429] = {X 342.9962, Y 49.6027, Z -6.3333, A 0.000, B 0.000, C 0.000 }
gfCNCPoint5[5430] = {X 340.9803, Y 49.2141, Z -6.3333, A 0.000, B 0.000, C 0.000 }
gfCNCPoint5[5431] = {X 339.0056, Y 48.6520, Z -6.3333, A 0.000, B 0.000, C 0.000 }
gfCNCPoint5[5432] = {X 337.0872, Y 47.9208, Z -6.3333, A 0.000, B 0.000, C 0.000 }
gfCNCPoint5[5433] = {X 335.2394, Y 47.0259, Z -6.3333, A 0.000, B 0.000, C 0.000 }
gfCNCPoint5[5434] = {X 333.6462, Y 46.0406, Z -6.3333, A 0.000, B 0.000, C 0.000 }
gfCNCPoint5[5435] = {X 332.1357, Y 44.9328, Z -6.3333, A 0.000, B 0.000, C 0.000 }
gfCNCPoint5[5436] = {X 330.7173, Y 43.7094, Z -6.3333, A 0.000, B 0.000, C 0.000 }
gfCNCPoint5[5437] = {X 329.7931, Y 43.7230, Z -6.3333, A 0.000, B 0.000, C 0.000 }
gfCNCPoint5[5438] = {X 328.8887, Y 43.5322, Z -6.3333, A 0.000, B 0.000, C 0.000 }
gfCNCPoint5[5439] = {X 328.0488, Y 43.1465, Z -6.3333, A 0.000, B 0.000, C 0.000 }
gfCNCPoint5[5440] = {X 327.3148, Y 42.5847, Z -6.3333, A 0.000, B 0.000, C 0.000 }
gfCNCPoint5[5441] = {X 326.6925, Y 41.9780, Z -6.3333, A 0.000, B 0.000, C 0.000 }
gfCNCPoint5[5442] = {X 326.0873, Y 41.2331, Z -6.3333, A 0.000, B 0.000, C 0.000 }
gfCNCPoint5[5443] = {X 325.6690, Y 40.3693, Z -6.3333, A 0.000, B 0.000, C 0.000 }
gfCNCPoint5[5444] = {X 325.4597, Y 39.4326, Z -6.3333, A 0.000, B 0.000, C 0.000 }
gfCNCPoint5[5445] = {X 325.4707, Y 38.4730, Z -6.3333, A 0.000, B 0.000, C 0.000 }
gfCNCPoint5[5446] = {X 325.7013, Y 37.5413, Z -6.3333, A 0.000, B 0.000, C 0.000 }
gfCNCPoint5[5447] = {X 326.1392, Y 36.6874, Z -6.3333, A 0.000, B 0.000, C 0.000 }
gfCNCPoint5[5448] = {X 330.3726, Y 30.3576, Z -6.3333, A 0.000, B 0.000, C 0.000 }
gfCNCPoint5[5449] = {X 330.9517, Y 29.6673, Z -6.3333, A 0.000, B 0.000, C 0.000 }
gfCNCPoint5[5450] = {X 331.6658, Y 29.1178, Z -6.3333, A 0.000, B 0.000, C 0.000 }
gfCNCPoint5[5451] = {X 332.4816, Y 28.7351, Z -6.3333, A 0.000, B 0.000, C 0.000 }
gfCNCPoint5[5452] = {X 333.3606, Y 28.5369, Z -6.3333, A 0.000, B 0.000, C 0.000 }
gfCNCPoint5[5453] = {X 334.2616, Y 28.5327, Z -6.3333, A 0.000, B 0.000, C 0.000 }
gfCNCPoint5[5454] = {X 335.1425, Y 28.7227, Z -6.3333, A 0.000, B 0.000, C 0.000 }
gfCNCPoint5[5455] = {X 335.9617, Y 29.0978, Z -6.3333, A 0.000, B 0.000, C 0.000 }
gfCNCPoint5[5456] = {X 336.6810, Y 29.6405, Z -6.3333, A 0.000, B 0.000, C 0.000 }
gfCNCPoint5[5457] = {X 337.3163, Y 30.2523, Z -6.3333, A 0.000, B 0.000, C 0.000 }
gfCNCPoint5[5458] = {X 337.8306, Y 30.8657, Z -6.3333, A 0.000, B 0.000, C 0.000 }
gfCNCPoint5[5459] = {X 338.2180, Y 31.5661, Z -6.3333, A 0.000, B 0.000, C 0.000 }
gfCNCPoint5[5460] = {X 338.4641, Y 32.3278, Z -6.3333, A 0.000, B 0.000, C 0.000 }
gfCNCPoint5[5461] = {X 338.5597, Y 33.1226, Z -6.3333, A 0.000, B 0.000, C 0.000 }
gfCNCPoint5[5462] = {X 338.5013, Y 33.9209, Z -6.3333, A 0.000, B 0.000, C 0.000 }
gfCNCPoint5[5463] = {X 339.1865, Y 34.5413, Z -6.3333, A 0.000, B 0.000, C 0.000 }
gfCNCPoint5[5464] = {X 339.8926, Y 35.1378, Z -6.3333, A 0.000, B 0.000, C 0.000 }
gfCNCPoint5[5465] = {X 341.0025, Y 35.9325, Z -6.3333, A 0.000, B 0.000, C 0.000 }
gfCNCPoint5[5466] = {X 342.2043, Y 36.5799, Z -6.3333, A 0.000, B 0.000, C 0.000 }
gfCNCPoint5[5467] = {X 343.4785, Y 37.0697, Z -6.3333, A 0.000, B 0.000, C 0.000 }
gfCNCPoint5[5468] = {X 344.8045, Y 37.3939, Z -6.3333, A 0.000, B 0.000, C 0.000 }
gfCNCPoint5[5469] = {X 346.1609, Y 37.5472, Z -6.3333, A 0.000, B 0.000, C 0.000 }
gfCNCPoint5[5470] = {X 347.5259, Y 37.5273, Z -6.3333, A 0.000, B 0.000, C 0.000 }
gfCNCPoint5[5471] = {X 348.7018, Y 37.3890, Z -6.3333, A 0.000, B 0.000, C 0.000 }
gfCNCPoint5[5472] = {X 349.8497, Y 37.0985, Z -6.3333, A 0.000, B 0.000, C 0.000 }
gfCNCPoint5[5473] = {X 350.9499, Y 36.6607, Z -6.3333, A 0.000, B 0.000, C 0.000 }
gfCNCPoint5[5474] = {X 351.9835, Y 36.0830, Z -6.3333, A 0.000, B 0.000, C 0.000 }
gfCNCPoint5[5475] = {X 352.9329, Y 35.3754, Z -6.3333, A 0.000, B 0.000, C 0.000 }
gfCNCPoint5[5476] = {X 354.1012, Y 34.2402, Z -6.3333, A 0.000, B 0.000, C 0.000 }
gfCNCPoint5[5477] = {X 355.1123, Y 32.9629, Z -6.3333, A 0.000, B 0.000, C 0.000 }
gfCNCPoint5[5478] = {X 355.9491, Y 31.5652, Z -6.3333, A 0.000, B 0.000, C 0.000 }
gfCNCPoint5[5479] = {X 356.5972, Y 30.0706, Z -6.3333, A 0.000, B 0.000, C 0.000 }
gfCNCPoint5[5480] = {X 357.0459, Y 28.5046, Z -6.3333, A 0.000, B 0.000, C 0.000 }
gfCNCPoint5[5481] = {X 357.3216, Y 26.8012, Z -6.3333, A 0.000, B 0.000, C 0.000 }
gfCNCPoint5[5482] = {X 357.4339, Y 25.0793, Z -6.3333, A 0.000, B 0.000, C 0.000 }
gfCNCPoint5[5483] = {X 357.3818, Y 23.3545, Z -6.3333, A 0.000, B 0.000, C 0.000 }
gfCNCPoint5[5484] = {X 357.1658, Y 21.6425, Z -6.3333, A 0.000, B 0.000, C 0.000 }
gfCNCPoint5[5485] = {X 356.8072, Y 20.1066, Z -6.3333, A 0.000, B 0.000, C 0.000 }
gfCNCPoint5[5486] = {X 356.2502, Y 18.6309, Z -6.3333, A 0.000, B 0.000, C 0.000 }
gfCNCPoint5[5487] = {X 355.5044, Y 17.2411, Z -6.3333, A 0.000, B 0.000, C 0.000 }
gfCNCPoint5[5488] = {X 354.5828, Y 15.9611, Z -6.3333, A 0.000, B 0.000, C 0.000 }
gfCNCPoint5[5489] = {X 353.6970, Y 15.0182, Z -6.3333, A 0.000, B 0.000, C 0.000 }
gfCNCPoint5[5490] = {X 352.6890, Y 14.2071, Z -6.3333, A 0.000, B 0.000, C 0.000 }
gfCNCPoint5[5491] = {X 351.5782, Y 13.5436, Z -6.3333, A 0.000, B 0.000, C 0.000 }
gfCNCPoint5[5492] = {X 350.3862, Y 13.0406, Z -6.3333, A 0.000, B 0.000, C 0.000 }
gfCNCPoint5[5493] = {X 349.1360, Y 12.7076, Z -6.3333, A 0.000, B 0.000, C 0.000 }
gfCNCPoint5[5494] = {X 347.5978, Y 12.5014, Z -6.3333, A 0.000, B 0.000, C 0.000 }
gfCNCPoint5[5495] = {X 346.0461, Y 12.4727, Z -6.3333, A 0.000, B 0.000, C 0.000 }
gfCNCPoint5[5496] = {X 344.5013, Y 12.6221, Z -6.3333, A 0.000, B 0.000, C 0.000 }
gfCNCPoint5[5497] = {X 342.9839, Y 12.9475, Z -6.3333, A 0.000, B 0.000, C 0.000 }
gfCNCPoint5[5498] = {X 341.5137, Y 13.4446, Z -6.3333, A 0.000, B 0.000, C 0.000 }
gfCNCPoint5[5499] = {X 340.1101, Y 14.1069, Z -6.3333, A 0.000, B 0.000, C 0.000 }
gfCNCPoint5[5500] = {X 338.7917, Y 14.9257, Z -6.3333, A 0.000, B 0.000, C 0.000 }
gfCNCPoint5[5501] = {X 338.7692, Y 15.7572, Z -6.3333, A 0.000, B 0.000, C 0.000 }
gfCNCPoint5[5502] = {X 338.5818, Y 16.5677, Z -6.3333, A 0.000, B 0.000, C 0.000 }
gfCNCPoint5[5503] = {X 338.2368, Y 17.3247, Z -6.3333, A 0.000, B 0.000, C 0.000 }
gfCNCPoint5[5504] = {X 337.7481, Y 17.9979, Z -6.3333, A 0.000, B 0.000, C 0.000 }
gfCNCPoint5[5505] = {X 337.1353, Y 18.5604, Z -6.3333, A 0.000, B 0.000, C 0.000 }
gfCNCPoint5[5506] = {X 336.4209, Y 19.0861, Z -6.3333, A 0.000, B 0.000, C 0.000 }
gfCNCPoint5[5507] = {X 335.6353, Y 19.5283, Z -6.3333, A 0.000, B 0.000, C 0.000 }
gfCNCPoint5[5508] = {X 334.7729, Y 19.7908, Z -6.3333, A 0.000, B 0.000, C 0.000 }
gfCNCPoint5[5509] = {X 333.8742, Y 19.8614, Z -6.3333, A 0.000, B 0.000, C 0.000 }
gfCNCPoint5[5510] = {X 332.9814, Y 19.7367, Z -6.3333, A 0.000, B 0.000, C 0.000 }
gfCNCPoint5[5511] = {X 332.1364, Y 19.4226, Z -6.3333, A 0.000, B 0.000, C 0.000 }
gfCNCPoint5[5512] = {X 331.3789, Y 18.9339, Z -6.3333, A 0.000, B 0.000, C 0.000 }
gfCNCPoint5[5513] = {X 330.7445, Y 18.2934, Z -6.3333, A 0.000, B 0.000, C 0.000 }
gfCNCPoint5[5514] = {X 330.2630, Y 17.5314, Z -6.3333, A 0.000, B 0.000, C 0.000 }
gfCNCPoint5[5515] = {X 326.7381, Y 10.2803, Z -6.3333, A 0.000, B 0.000, C 0.000 }
gfCNCPoint5[5516] = {X 326.4156, Y 9.3505, Z -6.3333, A 0.000, B 0.000, C 0.000 }
gfCNCPoint5[5517] = {X 326.3205, Y 8.3711, Z -6.3333, A 0.000, B 0.000, C 0.000 }
gfCNCPoint5[5518] = {X 326.4581, Y 7.3967, Z -6.3333, A 0.000, B 0.000, C 0.000 }
gfCNCPoint5[5519] = {X 326.8207, Y 6.4819, Z -6.3333, A 0.000, B 0.000, C 0.000 }
gfCNCPoint5[5520] = {X 327.3881, Y 5.6778, Z -6.3333, A 0.000, B 0.000, C 0.000 }
gfCNCPoint5[5521] = {X 328.1285, Y 5.0296, Z -6.3333, A 0.000, B 0.000, C 0.000 }
gfCNCPoint5[5522] = {X 328.7983, Y 4.5709, Z -6.3333, A 0.000, B 0.000, C 0.000 }
gfCNCPoint5[5523] = {X 329.6631, Y 4.1253, Z -6.3333, A 0.000, B 0.000, C 0.000 }
gfCNCPoint5[5524] = {X 330.6078, Y 3.8928, Z -6.3333, A 0.000, B 0.000, C 0.000 }
gfCNCPoint5[5525] = {X 331.5807, Y 3.8861, Z -6.3333, A 0.000, B 0.000, C 0.000 }
gfCNCPoint5[5526] = {X 332.5286, Y 4.1055, Z -6.3333, A 0.000, B 0.000, C 0.000 }
gfCNCPoint5[5527] = {X 334.2073, Y 3.1707, Z -6.3333, A 0.000, B 0.000, C 0.000 }
gfCNCPoint5[5528] = {X 335.9455, Y 2.3518, Z -6.3333, A 0.000, B 0.000, C 0.000 }
gfCNCPoint5[5529] = {X 338.0316, Y 1.5385, Z -6.3333, A 0.000, B 0.000, C 0.000 }
gfCNCPoint5[5530] = {X 340.1798, Y 0.9067, Z -6.3333, A 0.000, B 0.000, C 0.000 }
gfCNCPoint5[5531] = {X 342.3741, Y 0.4611, Z -6.3333, A 0.000, B 0.000, C 0.000 }
gfCNCPoint5[5532] = {X 344.5986, Y 0.2049, Z -6.3333, A 0.000, B 0.000, C 0.000 }
gfCNCPoint5[5533] = {X 346.8367, Y 0.1401, Z -6.3333, A 0.000, B 0.000, C 0.000 }
gfCNCPoint5[5534] = {X 349.0723, Y 0.2671, Z -6.3333, A 0.000, B 0.000, C 0.000 }
gfCNCPoint5[5535] = {X 351.2887, Y 0.5850, Z -6.3333, A 0.000, B 0.000, C 0.000 }
gfCNCPoint5[5536] = {X 351.5650, Y 0.6368, Z -6.3333, A 0.000, B 0.000, C 0.000 }
gfCNCPoint5[5537] = {X 352.3018, Y -3.2948, Z -6.3333, A 0.000, B 0.000, C 0.000 }
gfCNCPoint5[5538] = {X 351.5503, Y 0.7154, Z -6.3333, A 0.000, B 0.000, C 0.000 }
gfCNCPoint5[5539] = {X 351.8250, Y 0.7669, Z -6.3333, A 0.000, B 0.000, C 0.000 }
gfCNCPoint5[5540] = {X 353.7531, Y 1.2519, Z -6.3333, A 0.000, B 0.000, C 0.000 }
gfCNCPoint5[5541] = {X 355.6259, Y 1.9190, Z -6.3333, A 0.000, B 0.000, C 0.000 }
gfCNCPoint5[5542] = {X 357.4264, Y 2.7620, Z -6.3333, A 0.000, B 0.000, C 0.000 }
gfCNCPoint5[5543] = {X 359.1381, Y 3.7733, Z -6.3333, A 0.000, B 0.000, C 0.000 }
gfCNCPoint5[5544] = {X 360.7453, Y 4.9436, Z -6.3333, A 0.000, B 0.000, C 0.000 }
gfCNCPoint5[5545] = {X 362.2332, Y 6.2622, Z -6.3333, A 0.000, B 0.000, C 0.000 }
gfCNCPoint5[5546] = {X 363.5883, Y 7.7169, Z -6.3333, A 0.000, B 0.000, C 0.000 }
gfCNCPoint5[5547] = {X 364.9265, Y 9.4566, Z -6.3333, A 0.000, B 0.000, C 0.000 }
gfCNCPoint5[5548] = {X 366.1061, Y 11.3074, Z -6.3333, A 0.000, B 0.000, C 0.000 }
gfCNCPoint5[5549] = {X 367.1178, Y 13.2551, Z -6.3333, A 0.000, B 0.000, C 0.000 }
gfCNCPoint5[5550] = {X 367.9539, Y 15.2844, Z -6.3333, A 0.000, B 0.000, C 0.000 }
gfCNCPoint5[5551] = {X 368.6077, Y 17.3796, Z -6.3333, A 0.000, B 0.000, C 0.000 }
gfCNCPoint5[5552] = {X 369.0742, Y 19.5242, Z -6.3333, A 0.000, B 0.000, C 0.000 }
gfCNCPoint5[5553] = {X 369.4027, Y 21.8748, Z -6.3333, A 0.000, B 0.000, C 0.000 }
gfCNCPoint5[5554] = {X 369.5534, Y 24.2435, Z -6.3333, A 0.000, B 0.000, C 0.000 }
gfCNCPoint5[5555] = {X 369.5253, Y 26.6167, Z -6.3333, A 0.000, B 0.000, C 0.000 }
gfCNCPoint5[5556] = {X 369.3186, Y 28.9812, Z -6.3333, A 0.000, B 0.000, C 0.000 }
gfCNCPoint5[5557] = {X 368.9345, Y 31.3233, Z -6.3333, A 0.000, B 0.000, C 0.000 }
gfCNCPoint5[5558] = {X 368.4155, Y 33.4073, Z -6.3333, A 0.000, B 0.000, C 0.000 }
gfCNCPoint5[5559] = {X 367.7145, Y 35.4372, Z -6.3333, A 0.000, B 0.000, C 0.000 }
gfCNCPoint5[5560] = {X 366.8369, Y 37.3974, Z -6.3333, A 0.000, B 0.000, C 0.000 }
gfCNCPoint5[5561] = {X 365.7897, Y 39.2723, Z -6.3333, A 0.000, B 0.000, C 0.000 }
gfCNCPoint5[5562] = {X 364.5809, Y 41.0474, Z -6.3333, A 0.000, B 0.000, C 0.000 }
gfCNCPoint5[5563] = {X 364.4652, Y 41.2057, Z -6.3333, A 0.000, B 0.000, C 0.000 }
gfCNCPoint5[5564] = {X 363.0806, Y 42.8636, Z -6.3333, A 0.000, B 0.000, C 0.000 }
gfCNCPoint5[5565] = {X 361.5382, Y 44.3760, Z -6.3333, A 0.000, B 0.000, C 0.000 }
gfCNCPoint5[5566] = {X 359.8534, Y 45.7279, Z -6.3333, A 0.000, B 0.000, C 0.000 }
gfCNCPoint5[5567] = {X 358.0428, Y 46.9059, Z -6.3333, A 0.000, B 0.000, C 0.000 }
gfCNCPoint5[5568] = {X 356.1242, Y 47.8985, Z -6.3333, A 0.000, B 0.000, C 0.000 }
gfCNCPoint5[5569] = {X 353.9491, Y 48.7101, Z -6.3333, A 0.000, B 0.000, C 0.000 }
gfCNCPoint5[5570] = {X 351.7028, Y 49.2961, Z -6.3333, A 0.000, B 0.000, C 0.000 }
gfCNCPoint5[5571] = {X 349.4085, Y 49.6505, Z -6.3333, A 0.000, B 0.000, C 0.000 }
gfCNCPoint5[5572] = {X 347.0900, Y 49.7696, Z -6.3333, A 0.000, B 0.000, C 0.000 }
gfCNCPoint5[5573] = {X 345.0441, Y 49.7353, Z -6.3333, A 0.000, B 0.000, C 0.000 }
gfCNCPoint5[5574] = {X 343.0089, Y 49.5237, Z -6.3333, A 0.000, B 0.000, C 0.000 }
gfCNCPoint5[5575] = {X 340.9997, Y 49.1364, Z -6.3333, A 0.000, B 0.000, C 0.000 }
gfCNCPoint5[5576] = {X 339.0317, Y 48.5763, Z -6.3333, A 0.000, B 0.000, C 0.000 }
gfCNCPoint5[5577] = {X 337.1196, Y 47.8477, Z -6.3333, A 0.000, B 0.000, C 0.000 }
gfCNCPoint5[5578] = {X 335.2780, Y 46.9559, Z -6.3333, A 0.000, B 0.000, C 0.000 }
gfCNCPoint5[5579] = {X 333.6801, Y 45.9670, Z -6.3333, A 0.000, B 0.000, C 0.000 }
gfCNCPoint5[5580] = {X 332.1657, Y 44.8544, Z -6.3333, A 0.000, B 0.000, C 0.000 }
gfCNCPoint5[5581] = {X 330.7443, Y 43.6252, Z -6.3333, A 0.000, B 0.000, C 0.000 }
gfCNCPoint5[5582] = {X 329.8287, Y 43.6460, Z -6.3333, A 0.000, B 0.000, C 0.000 }
gfCNCPoint5[5583] = {X 328.9316, Y 43.4621, Z -6.3333, A 0.000, B 0.000, C 0.000 }
gfCNCPoint5[5584] = {X 328.0981, Y 43.0827, Z -6.3333, A 0.000, B 0.000, C 0.000 }
gfCNCPoint5[5585] = {X 327.3701, Y 42.5270, Z -6.3333, A 0.000, B 0.000, C 0.000 }
gfCNCPoint5[5586] = {X 326.7483, Y 41.9207, Z -6.3333, A 0.000, B 0.000, C 0.000 }
gfCNCPoint5[5587] = {X 326.1548, Y 41.1901, Z -6.3333, A 0.000, B 0.000, C 0.000 }
gfCNCPoint5[5588] = {X 325.7445, Y 40.3430, Z -6.3333, A 0.000, B 0.000, C 0.000 }
gfCNCPoint5[5589] = {X 325.5393, Y 39.4243, Z -6.3333, A 0.000, B 0.000, C 0.000 }
gfCNCPoint5[5590] = {X 325.5500, Y 38.4831, Z -6.3333, A 0.000, B 0.000, C 0.000 }
gfCNCPoint5[5591] = {X 325.7762, Y 37.5694, Z -6.3333, A 0.000, B 0.000, C 0.000 }
gfCNCPoint5[5592] = {X 326.2057, Y 36.7318, Z -6.3333, A 0.000, B 0.000, C 0.000 }
gfCNCPoint5[5593] = {X 330.4390, Y 30.4021, Z -6.3333, A 0.000, B 0.000, C 0.000 }
gfCNCPoint5[5594] = {X 331.0070, Y 29.7251, Z -6.3333, A 0.000, B 0.000, C 0.000 }
gfCNCPoint5[5595] = {X 331.7074, Y 29.1862, Z -6.3333, A 0.000, B 0.000, C 0.000 }
gfCNCPoint5[5596] = {X 332.5073, Y 28.8108, Z -6.3333, A 0.000, B 0.000, C 0.000 }
gfCNCPoint5[5597] = {X 333.3694, Y 28.6165, Z -6.3333, A 0.000, B 0.000, C 0.000 }
gfCNCPoint5[5598] = {X 334.2531, Y 28.6123, Z -6.3333, A 0.000, B 0.000, C 0.000 }
gfCNCPoint5[5599] = {X 335.1169, Y 28.7985, Z -6.3333, A 0.000, B 0.000, C 0.000 }
gfCNCPoint5[5600] = {X 335.9204, Y 29.1663, Z -6.3333, A 0.000, B 0.000, C 0.000 }
gfCNCPoint5[5601] = {X 336.6259, Y 29.6985, Z -6.3333, A 0.000, B 0.000, C 0.000 }
gfCNCPoint5[5602] = {X 337.2602, Y 30.3094, Z -6.3333, A 0.000, B 0.000, C 0.000 }
gfCNCPoint5[5603] = {X 337.7695, Y 30.9180, Z -6.3333, A 0.000, B 0.000, C 0.000 }
gfCNCPoint5[5604] = {X 338.1514, Y 31.6137, Z -6.3333, A 0.000, B 0.000, C 0.000 }
gfCNCPoint5[5605] = {X 338.3914, Y 32.3701, Z -6.3333, A 0.000, B 0.000, C 0.000 }
gfCNCPoint5[5606] = {X 338.4804, Y 33.1587, Z -6.3333, A 0.000, B 0.000, C 0.000 }
gfCNCPoint5[5607] = {X 338.4150, Y 33.9496, Z -6.3333, A 0.000, B 0.000, C 0.000 }
gfCNCPoint5[5608] = {X 339.1175, Y 34.5872, Z -6.3333, A 0.000, B 0.000, C 0.000 }
gfCNCPoint5[5609] = {X 339.8420, Y 35.1998, Z -6.3333, A 0.000, B 0.000, C 0.000 }
gfCNCPoint5[5610] = {X 340.9600, Y 36.0003, Z -6.3333, A 0.000, B 0.000, C 0.000 }
gfCNCPoint5[5611] = {X 342.1706, Y 36.6525, Z -6.3333, A 0.000, B 0.000, C 0.000 }
gfCNCPoint5[5612] = {X 343.4541, Y 37.1459, Z -6.3333, A 0.000, B 0.000, C 0.000 }
gfCNCPoint5[5613] = {X 344.7898, Y 37.4725, Z -6.3333, A 0.000, B 0.000, C 0.000 }
gfCNCPoint5[5614] = {X 346.1561, Y 37.6271, Z -6.3333, A 0.000, B 0.000, C 0.000 }
gfCNCPoint5[5615] = {X 347.5310, Y 37.6071, Z -6.3333, A 0.000, B 0.000, C 0.000 }
gfCNCPoint5[5616] = {X 348.7172, Y 37.4675, Z -6.3333, A 0.000, B 0.000, C 0.000 }
gfCNCPoint5[5617] = {X 349.8750, Y 37.1744, Z -6.3333, A 0.000, B 0.000, C 0.000 }
gfCNCPoint5[5618] = {X 350.9846, Y 36.7327, Z -6.3333, A 0.000, B 0.000, C 0.000 }
gfCNCPoint5[5619] = {X 352.0272, Y 36.1500, Z -6.3333, A 0.000, B 0.000, C 0.000 }
gfCNCPoint5[5620] = {X 352.9848, Y 35.4363, Z -6.3333, A 0.000, B 0.000, C 0.000 }
gfCNCPoint5[5621] = {X 354.1606, Y 34.2938, Z -6.3333, A 0.000, B 0.000, C 0.000 }
gfCNCPoint5[5622] = {X 355.1782, Y 33.0083, Z -6.3333, A 0.000, B 0.000, C 0.000 }
gfCNCPoint5[5623] = {X 356.0203, Y 31.6016, Z -6.3333, A 0.000, B 0.000, C 0.000 }
gfCNCPoint5[5624] = {X 356.6726, Y 30.0974, Z -6.3333, A 0.000, B 0.000, C 0.000 }
gfCNCPoint5[5625] = {X 357.1242, Y 28.5214, Z -6.3333, A 0.000, B 0.000, C 0.000 }
gfCNCPoint5[5626] = {X 357.4011, Y 26.8104, Z -6.3333, A 0.000, B 0.000, C 0.000 }
gfCNCPoint5[5627] = {X 357.5139, Y 25.0808, Z -6.3333, A 0.000, B 0.000, C 0.000 }
gfCNCPoint5[5628] = {X 357.4616, Y 23.3484, Z -6.3333, A 0.000, B 0.000, C 0.000 }
gfCNCPoint5[5629] = {X 357.2446, Y 21.6288, Z -6.3333, A 0.000, B 0.000, C 0.000 }
gfCNCPoint5[5630] = {X 356.8836, Y 20.0828, Z -6.3333, A 0.000, B 0.000, C 0.000 }
gfCNCPoint5[5631] = {X 356.3229, Y 18.5975, Z -6.3333, A 0.000, B 0.000, C 0.000 }
gfCNCPoint5[5632] = {X 355.5722, Y 17.1986, Z -6.3333, A 0.000, B 0.000, C 0.000 }
gfCNCPoint5[5633] = {X 354.6445, Y 15.9102, Z -6.3333, A 0.000, B 0.000, C 0.000 }
gfCNCPoint5[5634] = {X 353.7511, Y 14.9592, Z -6.3333, A 0.000, B 0.000, C 0.000 }
gfCNCPoint5[5635] = {X 352.7344, Y 14.1413, Z -6.3333, A 0.000, B 0.000, C 0.000 }
gfCNCPoint5[5636] = {X 351.6142, Y 13.4722, Z -6.3333, A 0.000, B 0.000, C 0.000 }
gfCNCPoint5[5637] = {X 350.4121, Y 12.9649, Z -6.3333, A 0.000, B 0.000, C 0.000 }
gfCNCPoint5[5638] = {X 349.1512, Y 12.6291, Z -6.3333, A 0.000, B 0.000, C 0.000 }
gfCNCPoint5[5639] = {X 347.5974, Y 12.4211, Z -6.3333, A 0.000, B 0.000, C 0.000 }
gfCNCPoint5[5640] = {X 346.0300, Y 12.3933, Z -6.3333, A 0.000, B 0.000, C 0.000 }
gfCNCPoint5[5641] = {X 344.4698, Y 12.5461, Z -6.3333, A 0.000, B 0.000, C 0.000 }
gfCNCPoint5[5642] = {X 342.9375, Y 12.8773, Z -6.3333, A 0.000, B 0.000, C 0.000 }
gfCNCPoint5[5643] = {X 341.4535, Y 13.3827, Z -6.3333, A 0.000, B 0.000, C 0.000 }
gfCNCPoint5[5644] = {X 340.0375, Y 14.0554, Z -6.3333, A 0.000, B 0.000, C 0.000 }
gfCNCPoint5[5645] = {X 338.7084, Y 14.8866, Z -6.3333, A 0.000, B 0.000, C 0.000 }
gfCNCPoint5[5646] = {X 338.6943, Y 15.7113, Z -6.3333, A 0.000, B 0.000, C 0.000 }
gfCNCPoint5[5647] = {X 338.5146, Y 16.5163, Z -6.3333, A 0.000, B 0.000, C 0.000 }
gfCNCPoint5[5648] = {X 338.1767, Y 17.2688, Z -6.3333, A 0.000, B 0.000, C 0.000 }
gfCNCPoint5[5649] = {X 337.6944, Y 17.9379, Z -6.3333, A 0.000, B 0.000, C 0.000 }
gfCNCPoint5[5650] = {X 337.0874, Y 18.4963, Z -6.3333, A 0.000, B 0.000, C 0.000 }
gfCNCPoint5[5651] = {X 336.3744, Y 19.0211, Z -6.3333, A 0.000, B 0.000, C 0.000 }
gfCNCPoint5[5652] = {X 335.6039, Y 19.4547, Z -6.3333, A 0.000, B 0.000, C 0.000 }
gfCNCPoint5[5653] = {X 334.7580, Y 19.7122, Z -6.3333, A 0.000, B 0.000, C 0.000 }
gfCNCPoint5[5654] = {X 333.8766, Y 19.7814, Z -6.3333, A 0.000, B 0.000, C 0.000 }
gfCNCPoint5[5655] = {X 333.0010, Y 19.6592, Z -6.3333, A 0.000, B 0.000, C 0.000 }
gfCNCPoint5[5656] = {X 332.1722, Y 19.3511, Z -6.3333, A 0.000, B 0.000, C 0.000 }
gfCNCPoint5[5657] = {X 331.4293, Y 18.8718, Z -6.3333, A 0.000, B 0.000, C 0.000 }
gfCNCPoint5[5658] = {X 330.8071, Y 18.2436, Z -6.3333, A 0.000, B 0.000, C 0.000 }
gfCNCPoint5[5659] = {X 330.3348, Y 17.4962, Z -6.3333, A 0.000, B 0.000, C 0.000 }
gfCNCPoint5[5660] = {X 326.8100, Y 10.2453, Z -6.3333, A 0.000, B 0.000, C 0.000 }
gfCNCPoint5[5661] = {X 326.4937, Y 9.3334, Z -6.3333, A 0.000, B 0.000, C 0.000 }
gfCNCPoint5[5662] = {X 326.4004, Y 8.3728, Z -6.3333, A 0.000, B 0.000, C 0.000 }
gfCNCPoint5[5663] = {X 326.5354, Y 7.4171, Z -6.3333, A 0.000, B 0.000, C 0.000 }
gfCNCPoint5[5664] = {X 326.8911, Y 6.5199, Z -6.3333, A 0.000, B 0.000, C 0.000 }
gfCNCPoint5[5665] = {X 327.4476, Y 5.7314, Z -6.3333, A 0.000, B 0.000, C 0.000 }
gfCNCPoint5[5666] = {X 328.1737, Y 5.0956, Z -6.3333, A 0.000, B 0.000, C 0.000 }
gfCNCPoint5[5667] = {X 328.8432, Y 4.6371, Z -6.3333, A 0.000, B 0.000, C 0.000 }
gfCNCPoint5[5668] = {X 329.7003, Y 4.1969, Z -6.3333, A 0.000, B 0.000, C 0.000 }
gfCNCPoint5[5669] = {X 330.6367, Y 3.9699, Z -6.3333, A 0.000, B 0.000, C 0.000 }
gfCNCPoint5[5670] = {X 331.6002, Y 3.9688, Z -6.3333, A 0.000, B 0.000, C 0.000 }
gfCNCPoint5[5671] = {X 332.5371, Y 4.1937, Z -6.3333, A 0.000, B 0.000, C 0.000 }
gfCNCPoint5[5672] = {X 334.2270, Y 3.2505, Z -6.3333, A 0.000, B 0.000, C 0.000 }
gfCNCPoint5[5673] = {X 335.9774, Y 2.4251, Z -6.3333, A 0.000, B 0.000, C 0.000 }
gfCNCPoint5[5674] = {X 338.0573, Y 1.6142, Z -6.3333, A 0.000, B 0.000, C 0.000 }
gfCNCPoint5[5675] = {X 340.1989, Y 0.9844, Z -6.3333, A 0.000, B 0.000, C 0.000 }
gfCNCPoint5[5676] = {X 342.3865, Y 0.5401, Z -6.3333, A 0.000, B 0.000, C 0.000 }
gfCNCPoint5[5677] = {X 344.6042, Y 0.2847, Z -6.3333, A 0.000, B 0.000, C 0.000 }
gfCNCPoint5[5678] = {X 346.8356, Y 0.2201, Z -6.3333, A 0.000, B 0.000, C 0.000 }
gfCNCPoint5[5679] = {X 349.0643, Y 0.3467, Z -6.3333, A 0.000, B 0.000, C 0.000 }
gfCNCPoint5[5680] = {X 351.2740, Y 0.6636, Z -6.3333, A 0.000, B 0.000, C 0.000 }
gfCNCPoint5[5681] = {X 351.5503, Y 0.7154, Z -6.3333, A 0.000, B 0.000, C 0.000 }
gfCNCPoint5[5682] = {X 352.2871, Y -3.2161, Z -6.3333, A 0.000, B 0.000, C 0.000 }
gfCNCPoint5[5683] = {X 351.5355, Y 0.7940, Z -6.3333, A 0.000, B 0.000, C 0.000 }
gfCNCPoint5[5684] = {X 351.8098, Y 0.8454, Z -6.3333, A 0.000, B 0.000, C 0.000 }
gfCNCPoint5[5685] = {X 353.7303, Y 1.3286, Z -6.3333, A 0.000, B 0.000, C 0.000 }
gfCNCPoint5[5686] = {X 355.5959, Y 1.9931, Z -6.3333, A 0.000, B 0.000, C 0.000 }
gfCNCPoint5[5687] = {X 357.3893, Y 2.8329, Z -6.3333, A 0.000, B 0.000, C 0.000 }
gfCNCPoint5[5688] = {X 359.0944, Y 3.8403, Z -6.3333, A 0.000, B 0.000, C 0.000 }
gfCNCPoint5[5689] = {X 360.6953, Y 5.0060, Z -6.3333, A 0.000, B 0.000, C 0.000 }
gfCNCPoint5[5690] = {X 362.1774, Y 6.3195, Z -6.3333, A 0.000, B 0.000, C 0.000 }
gfCNCPoint5[5691] = {X 363.5272, Y 7.7686, Z -6.3333, A 0.000, B 0.000, C 0.000 }
gfCNCPoint5[5692] = {X 364.8611, Y 9.5026, Z -6.3333, A 0.000, B 0.000, C 0.000 }
gfCNCPoint5[5693] = {X 366.0369, Y 11.3476, Z -6.3333, A 0.000, B 0.000, C 0.000 }
gfCNCPoint5[5694] = {X 367.0454, Y 13.2890, Z -6.3333, A 0.000, B 0.000, C 0.000 }
gfCNCPoint5[5695] = {X 367.8787, Y 15.3118, Z -6.3333, A 0.000, B 0.000, C 0.000 }
gfCNCPoint5[5696] = {X 368.5304, Y 17.4002, Z -6.3333, A 0.000, B 0.000, C 0.000 }
gfCNCPoint5[5697] = {X 368.9954, Y 19.5380, Z -6.3333, A 0.000, B 0.000, C 0.000 }
gfCNCPoint5[5698] = {X 369.3231, Y 21.8827, Z -6.3333, A 0.000, B 0.000, C 0.000 }
gfCNCPoint5[5699] = {X 369.4734, Y 24.2454, Z -6.3333, A 0.000, B 0.000, C 0.000 }
gfCNCPoint5[5700] = {X 369.4454, Y 26.6127, Z -6.3333, A 0.000, B 0.000, C 0.000 }
gfCNCPoint5[5701] = {X 369.2392, Y 28.9712, Z -6.3333, A 0.000, B 0.000, C 0.000 }
gfCNCPoint5[5702] = {X 368.8561, Y 31.3074, Z -6.3333, A 0.000, B 0.000, C 0.000 }
gfCNCPoint5[5703] = {X 368.3388, Y 33.3846, Z -6.3333, A 0.000, B 0.000, C 0.000 }
gfCNCPoint5[5704] = {X 367.6400, Y 35.4080, Z -6.3333, A 0.000, B 0.000, C 0.000 }
gfCNCPoint5[5705] = {X 366.7653, Y 37.3617, Z -6.3333, A 0.000, B 0.000, C 0.000 }
gfCNCPoint5[5706] = {X 365.7214, Y 39.2305, Z -6.3333, A 0.000, B 0.000, C 0.000 }
gfCNCPoint5[5707] = {X 364.5166, Y 40.9999, Z -6.3333, A 0.000, B 0.000, C 0.000 }
gfCNCPoint5[5708] = {X 364.4010, Y 41.1580, Z -6.3333, A 0.000, B 0.000, C 0.000 }
gfCNCPoint5[5709] = {X 363.1253, Y 42.6971, Z -6.3333, A 0.000, B 0.000, C 0.000 }
gfCNCPoint5[5710] = {X 361.7132, Y 44.1121, Z -6.3333, A 0.000, B 0.000, C 0.000 }
gfCNCPoint5[5711] = {X 360.1767, Y 45.3909, Z -6.3333, A 0.000, B 0.000, C 0.000 }
gfCNCPoint5[5712] = {X 358.5288, Y 46.5227, Z -6.3333, A 0.000, B 0.000, C 0.000 }
gfCNCPoint5[5713] = {X 356.7837, Y 47.4977, Z -6.3333, A 0.000, B 0.000, C 0.000 }
gfCNCPoint5[5714] = {X 356.0912, Y 47.8256, Z -6.3333, A 0.000, B 0.000, C 0.000 }
gfCNCPoint5[5715] = {X 353.9238, Y 48.6342, Z -6.3333, A 0.000, B 0.000, C 0.000 }
gfCNCPoint5[5716] = {X 351.6854, Y 49.2180, Z -6.3333, A 0.000, B 0.000, C 0.000 }
gfCNCPoint5[5717] = {X 349.3992, Y 49.5710, Z -6.3333, A 0.000, B 0.000, C 0.000 }
gfCNCPoint5[5718] = {X 347.0889, Y 49.6896, Z -6.3333, A 0.000, B 0.000, C 0.000 }
gfCNCPoint5[5719] = {X 345.0499, Y 49.6555, Z -6.3333, A 0.000, B 0.000, C 0.000 }
gfCNCPoint5[5720] = {X 343.0216, Y 49.4448, Z -6.3333, A 0.000, B 0.000, C 0.000 }
gfCNCPoint5[5721] = {X 341.0191, Y 49.0588, Z -6.3333, A 0.000, B 0.000, C 0.000 }
gfCNCPoint5[5722] = {X 339.0577, Y 48.5007, Z -6.3333, A 0.000, B 0.000, C 0.000 }
gfCNCPoint5[5723] = {X 337.1521, Y 47.7745, Z -6.3333, A 0.000, B 0.000, C 0.000 }
gfCNCPoint5[5724] = {X 335.3167, Y 46.8858, Z -6.3333, A 0.000, B 0.000, C 0.000 }
gfCNCPoint5[5725] = {X 333.7139, Y 45.8932, Z -6.3333, A 0.000, B 0.000, C 0.000 }
gfCNCPoint5[5726] = {X 332.1954, Y 44.7758, Z -6.3333, A 0.000, B 0.000, C 0.000 }
gfCNCPoint5[5727] = {X 330.7711, Y 43.5406, Z -6.3333, A 0.000, B 0.000, C 0.000 }
gfCNCPoint5[5728] = {X 329.8559, Y 43.5681, Z -6.3333, A 0.000, B 0.000, C 0.000 }
gfCNCPoint5[5729] = {X 328.9584, Y 43.3867, Z -6.3333, A 0.000, B 0.000, C 0.000 }
gfCNCPoint5[5730] = {X 328.1256, Y 43.0059, Z -6.3333, A 0.000, B 0.000, C 0.000 }
gfCNCPoint5[5731] = {X 327.4013, Y 42.4458, Z -6.3333, A 0.000, B 0.000, C 0.000 }
gfCNCPoint5[5732] = {X 326.8042, Y 41.8634, Z -6.3333, A 0.000, B 0.000, C 0.000 }
gfCNCPoint5[5733] = {X 326.2223, Y 41.1472, Z -6.3333, A 0.000, B 0.000, C 0.000 }
gfCNCPoint5[5734] = {X 325.8201, Y 40.3166, Z -6.3333, A 0.000, B 0.000, C 0.000 }
gfCNCPoint5[5735] = {X 325.6189, Y 39.4160, Z -6.3333, A 0.000, B 0.000, C 0.000 }
gfCNCPoint5[5736] = {X 325.6294, Y 38.4932, Z -6.3333, A 0.000, B 0.000, C 0.000 }
gfCNCPoint5[5737] = {X 325.8511, Y 37.5974, Z -6.3333, A 0.000, B 0.000, C 0.000 }
gfCNCPoint5[5738] = {X 326.2722, Y 36.7763, Z -6.3333, A 0.000, B 0.000, C 0.000 }
gfCNCPoint5[5739] = {X 330.5290, Y 30.4119, Z -6.3333, A 0.000, B 0.000, C 0.000 }
gfCNCPoint5[5740] = {X 331.0932, Y 29.7536, Z -6.3333, A 0.000, B 0.000, C 0.000 }
gfCNCPoint5[5741] = {X 331.7861, Y 29.2322, Z -6.3333, A 0.000, B 0.000, C 0.000 }
gfCNCPoint5[5742] = {X 332.5750, Y 28.8724, Z -6.3333, A 0.000, B 0.000, C 0.000 }
gfCNCPoint5[5743] = {X 333.4229, Y 28.6911, Z -6.3333, A 0.000, B 0.000, C 0.000 }
gfCNCPoint5[5744] = {X 334.2900, Y 28.6968, Z -6.3333, A 0.000, B 0.000, C 0.000 }
gfCNCPoint5[5745] = {X 335.1355, Y 28.8892, Z -6.3333, A 0.000, B 0.000, C 0.000 }
gfCNCPoint5[5746] = {X 335.9196, Y 29.2593, Z -6.3333, A 0.000, B 0.000, C 0.000 }
gfCNCPoint5[5747] = {X 336.6056, Y 29.7896, Z -6.3333, A 0.000, B 0.000, C 0.000 }
gfCNCPoint5[5748] = {X 337.2041, Y 30.3665, Z -6.3333, A 0.000, B 0.000, C 0.000 }
gfCNCPoint5[5749] = {X 337.7083, Y 30.9703, Z -6.3333, A 0.000, B 0.000, C 0.000 }
gfCNCPoint5[5750] = {X 338.0846, Y 31.6611, Z -6.3333, A 0.000, B 0.000, C 0.000 }
gfCNCPoint5[5751] = {X 338.3184, Y 32.4122, Z -6.3333, A 0.000, B 0.000, C 0.000 }
gfCNCPoint5[5752] = {X 338.4007, Y 33.1945, Z -6.3333, A 0.000, B 0.000, C 0.000 }
gfCNCPoint5[5753] = {X 338.3283, Y 33.9779, Z -6.3333, A 0.000, B 0.000, C 0.000 }
gfCNCPoint5[5754] = {X 339.0484, Y 34.6329, Z -6.3333, A 0.000, B 0.000, C 0.000 }
gfCNCPoint5[5755] = {X 339.7914, Y 35.2618, Z -6.3333, A 0.000, B 0.000, C 0.000 }
gfCNCPoint5[5756] = {X 341.1047, Y 36.1813, Z -6.3333, A 0.000, B 0.000, C 0.000 }
gfCNCPoint5[5757] = {X 342.5387, Y 36.8982, Z -6.3333, A 0.000, B 0.000, C 0.000 }
gfCNCPoint5[5758] = {X 344.0624, Y 37.3970, Z -6.3333, A 0.000, B 0.000, C 0.000 }
gfCNCPoint5[5759] = {X 345.6427, Y 37.6669, Z -6.3333, A 0.000, B 0.000, C 0.000 }
gfCNCPoint5[5760] = {X 347.2456, Y 37.7020, Z -6.3333, A 0.000, B 0.000, C 0.000 }
gfCNCPoint5[5761] = {X 347.5352, Y 37.6870, Z -6.3333, A 0.000, B 0.000, C 0.000 }
gfCNCPoint5[5762] = {X 348.7317, Y 37.5462, Z -6.3333, A 0.000, B 0.000, C 0.000 }
gfCNCPoint5[5763] = {X 349.8996, Y 37.2505, Z -6.3333, A 0.000, B 0.000, C 0.000 }
gfCNCPoint5[5764] = {X 351.0190, Y 36.8050, Z -6.3333, A 0.000, B 0.000, C 0.000 }
gfCNCPoint5[5765] = {X 352.0707, Y 36.2172, Z -6.3333, A 0.000, B 0.000, C 0.000 }
gfCNCPoint5[5766] = {X 353.0367, Y 35.4972, Z -6.3333, A 0.000, B 0.000, C 0.000 }
gfCNCPoint5[5767] = {X 354.2200, Y 34.3474, Z -6.3333, A 0.000, B 0.000, C 0.000 }
gfCNCPoint5[5768] = {X 355.2441, Y 33.0537, Z -6.3333, A 0.000, B 0.000, C 0.000 }
gfCNCPoint5[5769] = {X 356.0915, Y 31.6380, Z -6.3333, A 0.000, B 0.000, C 0.000 }
gfCNCPoint5[5770] = {X 356.7480, Y 30.1243, Z -6.3333, A 0.000, B 0.000, C 0.000 }
gfCNCPoint5[5771] = {X 357.2024, Y 28.5381, Z -6.3333, A 0.000, B 0.000, C 0.000 }
gfCNCPoint5[5772] = {X 357.4806, Y 26.8196, Z -6.3333, A 0.000, B 0.000, C 0.000 }
gfCNCPoint5[5773] = {X 357.5939, Y 25.0823, Z -6.3333, A 0.000, B 0.000, C 0.000 }
gfCNCPoint5[5774] = {X 357.5414, Y 23.3422, Z -6.3333, A 0.000, B 0.000, C 0.000 }
gfCNCPoint5[5775] = {X 357.3234, Y 21.6150, Z -6.3333, A 0.000, B 0.000, C 0.000 }
gfCNCPoint5[5776] = {X 356.9599, Y 20.0589, Z -6.3333, A 0.000, B 0.000, C 0.000 }
gfCNCPoint5[5777] = {X 356.3955, Y 18.5640, Z -6.3333, A 0.000, B 0.000, C 0.000 }
gfCNCPoint5[5778] = {X 355.6400, Y 17.1560, Z -6.3333, A 0.000, B 0.000, C 0.000 }
gfCNCPoint5[5779] = {X 354.7062, Y 15.8593, Z -6.3333, A 0.000, B 0.000, C 0.000 }
gfCNCPoint5[5780] = {X 353.8052, Y 14.9003, Z -6.3333, A 0.000, B 0.000, C 0.000 }
gfCNCPoint5[5781] = {X 352.7799, Y 14.0755, Z -6.3333, A 0.000, B 0.000, C 0.000 }
gfCNCPoint5[5782] = {X 351.6502, Y 13.4008, Z -6.3333, A 0.000, B 0.000, C 0.000 }
gfCNCPoint5[5783] = {X 350.4379, Y 12.8891, Z -6.3333, A 0.000, B 0.000, C 0.000 }
gfCNCPoint5[5784] = {X 349.1664, Y 12.5505, Z -6.3333, A 0.000, B 0.000, C 0.000 }
gfCNCPoint5[5785] = {X 347.3712, Y 12.3258, Z -6.3333, A 0.000, B 0.000, C 0.000 }
gfCNCPoint5[5786] = {X 345.5620, Y 12.3399, Z -6.3333, A 0.000, B 0.000, C 0.000 }
gfCNCPoint5[5787] = {X 343.7706, Y 12.5926, Z -6.3333, A 0.000, B 0.000, C 0.000 }
gfCNCPoint5[5788] = {X 342.0281, Y 13.0794, Z -6.3333, A 0.000, B 0.000, C 0.000 }
gfCNCPoint5[5789] = {X 340.3651, Y 13.7919, Z -6.3333, A 0.000, B 0.000, C 0.000 }
gfCNCPoint5[5790] = {X 338.8107, Y 14.7175, Z -6.3333, A 0.000, B 0.000, C 0.000 }
gfCNCPoint5[5791] = {X 338.7180, Y 14.7819, Z -6.3333, A 0.000, B 0.000, C 0.000 }
gfCNCPoint5[5792] = {X 338.6259, Y 14.8470, Z -6.3333, A 0.000, B 0.000, C 0.000 }
gfCNCPoint5[5793] = {X 338.6379, Y 15.0636, Z -6.3333, A 0.000, B 0.000, C 0.000 }
gfCNCPoint5[5794] = {X 338.5596, Y 16.0359, Z -6.3333, A 0.000, B 0.000, C 0.000 }
gfCNCPoint5[5795] = {X 338.2482, Y 16.9603, Z -6.3333, A 0.000, B 0.000, C 0.000 }
gfCNCPoint5[5796] = {X 337.7223, Y 17.7819, Z -6.3333, A 0.000, B 0.000, C 0.000 }
gfCNCPoint5[5797] = {X 337.0132, Y 18.4517, Z -6.3333, A 0.000, B 0.000, C 0.000 }
gfCNCPoint5[5798] = {X 336.3278, Y 18.9560, Z -6.3333, A 0.000, B 0.000, C 0.000 }
gfCNCPoint5[5799] = {X 335.5713, Y 19.3817, Z -6.3333, A 0.000, B 0.000, C 0.000 }
gfCNCPoint5[5800] = {X 334.7407, Y 19.6341, Z -6.3333, A 0.000, B 0.000, C 0.000 }
gfCNCPoint5[5801] = {X 333.8753, Y 19.7014, Z -6.3333, A 0.000, B 0.000, C 0.000 }
gfCNCPoint5[5802] = {X 333.0157, Y 19.5804, Z -6.3333, A 0.000, B 0.000, C 0.000 }
gfCNCPoint5[5803] = {X 332.2025, Y 19.2768, Z -6.3333, A 0.000, B 0.000, C 0.000 }
gfCNCPoint5[5804] = {X 331.4739, Y 18.8049, Z -6.3333, A 0.000, B 0.000, C 0.000 }
gfCNCPoint5[5805] = {X 330.8643, Y 18.1870, Z -6.3333, A 0.000, B 0.000, C 0.000 }
gfCNCPoint5[5806] = {X 330.4023, Y 17.4521, Z -6.3333, A 0.000, B 0.000, C 0.000 }
gfCNCPoint5[5807] = {X 326.8820, Y 10.2103, Z -6.3333, A 0.000, B 0.000, C 0.000 }
gfCNCPoint5[5808] = {X 326.5719, Y 9.3163, Z -6.3333, A 0.000, B 0.000, C 0.000 }
gfCNCPoint5[5809] = {X 326.4804, Y 8.3746, Z -6.3333, A 0.000, B 0.000, C 0.000 }
gfCNCPoint5[5810] = {X 326.6127, Y 7.4376, Z -6.3333, A 0.000, B 0.000, C 0.000 }
gfCNCPoint5[5811] = {X 326.9614, Y 6.5580, Z -6.3333, A 0.000, B 0.000, C 0.000 }
gfCNCPoint5[5812] = {X 327.5070, Y 5.7849, Z -6.3333, A 0.000, B 0.000, C 0.000 }
gfCNCPoint5[5813] = {X 328.2189, Y 5.1616, Z -6.3333, A 0.000, B 0.000, C 0.000 }
gfCNCPoint5[5814] = {X 328.8880, Y 4.7034, Z -6.3333, A 0.000, B 0.000, C 0.000 }
gfCNCPoint5[5815] = {X 329.7043, Y 4.2813, Z -6.3333, A 0.000, B 0.000, C 0.000 }
gfCNCPoint5[5816] = {X 330.5954, Y 4.0567, Z -6.3333, A 0.000, B 0.000, C 0.000 }
gfCNCPoint5[5817] = {X 331.5142, Y 4.0413, Z -6.3333, A 0.000, B 0.000, C 0.000 }
gfCNCPoint5[5818] = {X 332.4122, Y 4.2361, Z -6.3333, A 0.000, B 0.000, C 0.000 }
gfCNCPoint5[5819] = {X 332.5467, Y 4.2814, Z -6.3333, A 0.000, B 0.000, C 0.000 }
gfCNCPoint5[5820] = {X 332.6254, Y 4.2340, Z -6.3333, A 0.000, B 0.000, C 0.000 }
gfCNCPoint5[5821] = {X 332.7041, Y 4.1868, Z -6.3333, A 0.000, B 0.000, C 0.000 }
gfCNCPoint5[5822] = {X 334.3288, Y 3.2883, Z -6.3333, A 0.000, B 0.000, C 0.000 }
gfCNCPoint5[5823] = {X 336.0092, Y 2.4986, Z -6.3333, A 0.000, B 0.000, C 0.000 }
gfCNCPoint5[5824] = {X 336.1737, Y 2.4275, Z -6.3333, A 0.000, B 0.000, C 0.000 }
gfCNCPoint5[5825] = {X 338.2284, Y 1.6414, Z -6.3333, A 0.000, B 0.000, C 0.000 }
gfCNCPoint5[5826] = {X 340.3422, Y 1.0320, Z -6.3333, A 0.000, B 0.000, C 0.000 }
gfCNCPoint5[5827] = {X 342.5001, Y 0.6036, Z -6.3333, A 0.000, B 0.000, C 0.000 }
gfCNCPoint5[5828] = {X 344.6864, Y 0.3594, Z -6.3333, A 0.000, B 0.000, C 0.000 }
gfCNCPoint5[5829] = {X 346.8855, Y 0.3010, Z -6.3333, A 0.000, B 0.000, C 0.000 }
gfCNCPoint5[5830] = {X 349.0817, Y 0.4290, Z -6.3333, A 0.000, B 0.000, C 0.000 }
gfCNCPoint5[5831] = {X 351.2592, Y 0.7423, Z -6.3333, A 0.000, B 0.000, C 0.000 }
gfCNCPoint5[5832] = {X 351.5355, Y 0.7940, Z -6.3333, A 0.000, B 0.000, C 0.000 }
gfCNCPoint5[5833] = {X 352.2871, Y -3.2161, Z -6.3333, A 0.000, B 0.000, C 0.000 }
gfCNCPoint5[5834] = {X 352.2871, Y -3.2161, Z -3.3333, A 0.000, B 0.000, C 0.000 }
gfCNCPoint5[5835] = {X 352.2871, Y -3.2161, Z 11.0000, A 0.000, B 0.000, C 0.000 }
gfCNCPoint5[5836] = {X 606.0426, Y 42.9005, Z 11.0000, A 0.000, B 0.000, C 0.000 }
gfCNCPoint5[5837] = {X 606.0426, Y 42.9005, Z -3.3333, A 0.000, B 0.000, C 0.000 }
gfCNCPoint5[5838] = {X 606.0426, Y 42.9005, Z -6.3333, A 0.000, B 0.000, C 0.000 }
gfCNCPoint5[5839] = {X 603.6966, Y 47.0767, Z -6.3333, A 0.000, B 0.000, C 0.000 }
gfCNCPoint5[5840] = {X 603.6311, Y 47.1892, Z -6.3333, A 0.000, B 0.000, C 0.000 }
gfCNCPoint5[5841] = {X 603.5622, Y 47.2996, Z -6.3333, A 0.000, B 0.000, C 0.000 }
gfCNCPoint5[5842] = {X 603.0358, Y 47.9600, Z -6.3333, A 0.000, B 0.000, C 0.000 }
gfCNCPoint5[5843] = {X 602.3889, Y 48.5029, Z -6.3333, A 0.000, B 0.000, C 0.000 }
gfCNCPoint5[5844] = {X 601.6473, Y 48.9069, Z -6.3333, A 0.000, B 0.000, C 0.000 }
gfCNCPoint5[5845] = {X 600.8403, Y 49.1559, Z -6.3333, A 0.000, B 0.000, C 0.000 }
gfCNCPoint5[5846] = {X 600.0000, Y 49.2400, Z -6.3333, A 0.000, B 0.000, C 0.000 }
gfCNCPoint5[5847] = {X 593.5565, Y 49.2400, Z -6.3333, A 0.000, B 0.000, C 0.000 }
gfCNCPoint5[5848] = {X 592.6130, Y 49.1337, Z -6.3333, A 0.000, B 0.000, C 0.000 }
gfCNCPoint5[5849] = {X 591.7169, Y 48.8201, Z -6.3333, A 0.000, B 0.000, C 0.000 }
gfCNCPoint5[5850] = {X 590.9129, Y 48.3150, Z -6.3333, A 0.000, B 0.000, C 0.000 }
gfCNCPoint5[5851] = {X 590.2416, Y 47.6436, Z -6.3333, A 0.000, B 0.000, C 0.000 }
gfCNCPoint5[5852] = {X 589.7364, Y 46.8397, Z -6.3333, A 0.000, B 0.000, C 0.000 }
gfCNCPoint5[5853] = {X 589.4228, Y 45.9435, Z -6.3333, A 0.000, B 0.000, C 0.000 }
gfCNCPoint5[5854] = {X 589.3165, Y 45.0000, Z -6.3333, A 0.000, B 0.000, C 0.000 }
gfCNCPoint5[5855] = {X 589.3165, Y 44.0650, Z -6.3333, A 0.000, B 0.000, C 0.000 }
gfCNCPoint5[5856] = {X 589.4206, Y 43.1447, Z -6.3333, A 0.000, B 0.000, C 0.000 }
gfCNCPoint5[5857] = {X 589.7202, Y 42.2684, Z -6.3333, A 0.000, B 0.000, C 0.000 }
gfCNCPoint5[5858] = {X 590.2014, Y 41.4772, Z -6.3333, A 0.000, B 0.000, C 0.000 }
gfCNCPoint5[5859] = {X 590.8416, Y 40.8080, Z -6.3333, A 0.000, B 0.000, C 0.000 }
gfCNCPoint5[5860] = {X 590.8423, Y 33.1217, Z -6.3333, A 0.000, B 0.000, C 0.000 }
gfCNCPoint5[5861] = {X 585.3714, Y 46.6218, Z -6.3333, A 0.000, B 0.000, C 0.000 }
gfCNCPoint5[5862] = {X 585.0085, Y 47.3114, Z -6.3333, A 0.000, B 0.000, C 0.000 }
gfCNCPoint5[5863] = {X 584.5255, Y 47.9228, Z -6.3333, A 0.000, B 0.000, C 0.000 }
gfCNCPoint5[5864] = {X 583.9387, Y 48.4356, Z -6.3333, A 0.000, B 0.000, C 0.000 }
gfCNCPoint5[5865] = {X 583.2680, Y 48.8323, Z -6.3333, A 0.000, B 0.000, C 0.000 }
gfCNCPoint5[5866] = {X 582.3418, Y 49.1460, Z -6.3333, A 0.000, B 0.000, C 0.000 }
gfCNCPoint5[5867] = {X 581.3682, Y 49.2391, Z -6.3333, A 0.000, B 0.000, C 0.000 }
gfCNCPoint5[5868] = {X 580.3993, Y 49.1068, Z -6.3333, A 0.000, B 0.000, C 0.000 }
gfCNCPoint5[5869] = {X 579.4864, Y 48.7559, Z -6.3333, A 0.000, B 0.000, C 0.000 }
gfCNCPoint5[5870] = {X 578.6782, Y 48.2052, Z -6.3333, A 0.000, B 0.000, C 0.000 }
gfCNCPoint5[5871] = {X 578.0177, Y 47.4840, Z -6.3333, A 0.000, B 0.000, C 0.000 }
gfCNCPoint5[5872] = {X 577.5400, Y 46.6307, Z -6.3333, A 0.000, B 0.000, C 0.000 }
gfCNCPoint5[5873] = {X 571.9395, Y 32.9361, Z -6.3333, A 0.000, B 0.000, C 0.000 }
gfCNCPoint5[5874] = {X 571.9398, Y 40.8084, Z -6.3333, A 0.000, B 0.000, C 0.000 }
gfCNCPoint5[5875] = {X 571.9712, Y 40.8342, Z -6.3333, A 0.000, B 0.000, C 0.000 }
gfCNCPoint5[5876] = {X 572.5962, Y 41.4926, Z -6.3333, A 0.000, B 0.000, C 0.000 }
gfCNCPoint5[5877] = {X 573.0668, Y 42.2690, Z -6.3333, A 0.000, B 0.000, C 0.000 }
gfCNCPoint5[5878] = {X 573.3613, Y 43.1277, Z -6.3333, A 0.000, B 0.000, C 0.000 }
gfCNCPoint5[5879] = {X 573.4663, Y 44.0294, Z -6.3333, A 0.000, B 0.000, C 0.000 }
gfCNCPoint5[5880] = {X 573.4664, Y 45.0000, Z -6.3333, A 0.000, B 0.000, C 0.000 }
gfCNCPoint5[5881] = {X 573.3601, Y 45.9435, Z -6.3333, A 0.000, B 0.000, C 0.000 }
gfCNCPoint5[5882] = {X 573.0465, Y 46.8397, Z -6.3333, A 0.000, B 0.000, C 0.000 }
gfCNCPoint5[5883] = {X 572.5414, Y 47.6436, Z -6.3333, A 0.000, B 0.000, C 0.000 }
gfCNCPoint5[5884] = {X 571.8700, Y 48.3150, Z -6.3333, A 0.000, B 0.000, C 0.000 }
gfCNCPoint5[5885] = {X 571.0661, Y 48.8201, Z -6.3333, A 0.000, B 0.000, C 0.000 }
gfCNCPoint5[5886] = {X 570.1699, Y 49.1337, Z -6.3333, A 0.000, B 0.000, C 0.000 }
gfCNCPoint5[5887] = {X 569.2264, Y 49.2400, Z -6.3333, A 0.000, B 0.000, C 0.000 }
gfCNCPoint5[5888] = {X 562.4443, Y 49.2400, Z -6.3333, A 0.000, B 0.000, C 0.000 }
gfCNCPoint5[5889] = {X 561.5008, Y 49.1337, Z -6.3333, A 0.000, B 0.000, C 0.000 }
gfCNCPoint5[5890] = {X 560.6046, Y 48.8201, Z -6.3333, A 0.000, B 0.000, C 0.000 }
gfCNCPoint5[5891] = {X 559.8007, Y 48.3150, Z -6.3333, A 0.000, B 0.000, C 0.000 }
gfCNCPoint5[5892] = {X 559.1293, Y 47.6436, Z -6.3333, A 0.000, B 0.000, C 0.000 }
gfCNCPoint5[5893] = {X 558.6242, Y 46.8397, Z -6.3333, A 0.000, B 0.000, C 0.000 }
gfCNCPoint5[5894] = {X 558.3106, Y 45.9435, Z -6.3333, A 0.000, B 0.000, C 0.000 }
gfCNCPoint5[5895] = {X 558.2043, Y 45.0000, Z -6.3333, A 0.000, B 0.000, C 0.000 }
gfCNCPoint5[5896] = {X 558.2043, Y 44.0651, Z -6.3333, A 0.000, B 0.000, C 0.000 }
gfCNCPoint5[5897] = {X 558.3081, Y 43.1444, Z -6.3333, A 0.000, B 0.000, C 0.000 }
gfCNCPoint5[5898] = {X 558.6080, Y 42.2678, Z -6.3333, A 0.000, B 0.000, C 0.000 }
gfCNCPoint5[5899] = {X 559.0900, Y 41.4765, Z -6.3333, A 0.000, B 0.000, C 0.000 }
gfCNCPoint5[5900] = {X 559.7312, Y 40.8077, Z -6.3333, A 0.000, B 0.000, C 0.000 }
gfCNCPoint5[5901] = {X 559.7312, Y 9.1924, Z -6.3333, A 0.000, B 0.000, C 0.000 }
gfCNCPoint5[5902] = {X 559.0935, Y 8.5321, Z -6.3333, A 0.000, B 0.000, C 0.000 }
gfCNCPoint5[5903] = {X 558.6128, Y 7.7500, Z -6.3333, A 0.000, B 0.000, C 0.000 }
gfCNCPoint5[5904] = {X 558.3118, Y 6.8828, Z -6.3333, A 0.000, B 0.000, C 0.000 }
gfCNCPoint5[5905] = {X 558.2045, Y 5.9711, Z -6.3333, A 0.000, B 0.000, C 0.000 }
gfCNCPoint5[5906] = {X 558.2043, Y 5.0000, Z -6.3333, A 0.000, B 0.000, C 0.000 }
gfCNCPoint5[5907] = {X 558.3106, Y 4.0565, Z -6.3333, A 0.000, B 0.000, C 0.000 }
gfCNCPoint5[5908] = {X 558.6242, Y 3.1603, Z -6.3333, A 0.000, B 0.000, C 0.000 }
gfCNCPoint5[5909] = {X 559.1293, Y 2.3564, Z -6.3333, A 0.000, B 0.000, C 0.000 }
gfCNCPoint5[5910] = {X 559.8007, Y 1.6850, Z -6.3333, A 0.000, B 0.000, C 0.000 }
gfCNCPoint5[5911] = {X 560.6046, Y 1.1799, Z -6.3333, A 0.000, B 0.000, C 0.000 }
gfCNCPoint5[5912] = {X 561.5008, Y 0.8663, Z -6.3333, A 0.000, B 0.000, C 0.000 }
gfCNCPoint5[5913] = {X 562.4443, Y 0.7600, Z -6.3333, A 0.000, B 0.000, C 0.000 }
gfCNCPoint5[5914] = {X 570.9376, Y 0.7600, Z -6.3333, A 0.000, B 0.000, C 0.000 }
gfCNCPoint5[5915] = {X 571.8810, Y 0.8663, Z -6.3333, A 0.000, B 0.000, C 0.000 }
gfCNCPoint5[5916] = {X 572.7772, Y 1.1799, Z -6.3333, A 0.000, B 0.000, C 0.000 }
gfCNCPoint5[5917] = {X 573.5812, Y 1.6850, Z -6.3333, A 0.000, B 0.000, C 0.000 }
gfCNCPoint5[5918] = {X 574.2525, Y 2.3564, Z -6.3333, A 0.000, B 0.000, C 0.000 }
gfCNCPoint5[5919] = {X 574.7577, Y 3.1603, Z -6.3333, A 0.000, B 0.000, C 0.000 }
gfCNCPoint5[5920] = {X 575.0712, Y 4.0565, Z -6.3333, A 0.000, B 0.000, C 0.000 }
gfCNCPoint5[5921] = {X 575.1776, Y 5.0000, Z -6.3333, A 0.000, B 0.000, C 0.000 }
gfCNCPoint5[5922] = {X 575.1776, Y 5.9342, Z -6.3333, A 0.000, B 0.000, C 0.000 }
gfCNCPoint5[5923] = {X 575.1024, Y 6.7289, Z -6.3333, A 0.000, B 0.000, C 0.000 }
gfCNCPoint5[5924] = {X 574.8797, Y 7.4953, Z -6.3333, A 0.000, B 0.000, C 0.000 }
gfCNCPoint5[5925] = {X 574.5172, Y 8.2064, Z -6.3333, A 0.000, B 0.000, C 0.000 }
gfCNCPoint5[5926] = {X 581.1908, Y 24.5808, Z -6.3333, A 0.000, B 0.000, C 0.000 }
gfCNCPoint5[5927] = {X 587.9346, Y 8.0876, Z -6.3333, A 0.000, B 0.000, C 0.000 }
gfCNCPoint5[5928] = {X 587.6157, Y 7.4197, Z -6.3333, A 0.000, B 0.000, C 0.000 }
gfCNCPoint5[5929] = {X 587.4179, Y 6.7065, Z -6.3333, A 0.000, B 0.000, C 0.000 }
gfCNCPoint5[5930] = {X 587.3471, Y 5.9698, Z -6.3333, A 0.000, B 0.000, C 0.000 }
gfCNCPoint5[5931] = {X 587.3470, Y 5.0000, Z -6.3333, A 0.000, B 0.000, C 0.000 }
gfCNCPoint5[5932] = {X 587.4533, Y 4.0565, Z -6.3333, A 0.000, B 0.000, C 0.000 }
gfCNCPoint5[5933] = {X 587.7668, Y 3.1603, Z -6.3333, A 0.000, B 0.000, C 0.000 }
gfCNCPoint5[5934] = {X 588.2720, Y 2.3564, Z -6.3333, A 0.000, B 0.000, C 0.000 }
gfCNCPoint5[5935] = {X 588.9434, Y 1.6850, Z -6.3333, A 0.000, B 0.000, C 0.000 }
gfCNCPoint5[5936] = {X 589.7473, Y 1.1799, Z -6.3333, A 0.000, B 0.000, C 0.000 }
gfCNCPoint5[5937] = {X 590.6435, Y 0.8663, Z -6.3333, A 0.000, B 0.000, C 0.000 }
gfCNCPoint5[5938] = {X 591.5870, Y 0.7600, Z -6.3333, A 0.000, B 0.000, C 0.000 }
gfCNCPoint5[5939] = {X 600.0000, Y 0.7600, Z -6.3333, A 0.000, B 0.000, C 0.000 }
gfCNCPoint5[5940] = {X 600.8403, Y 0.8441, Z -6.3333, A 0.000, B 0.000, C 0.000 }
gfCNCPoint5[5941] = {X 601.6473, Y 1.0931, Z -6.3333, A 0.000, B 0.000, C 0.000 }
gfCNCPoint5[5942] = {X 602.3889, Y 1.4971, Z -6.3333, A 0.000, B 0.000, C 0.000 }
gfCNCPoint5[5943] = {X 603.0358, Y 2.0400, Z -6.3333, A 0.000, B 0.000, C 0.000 }
gfCNCPoint5[5944] = {X 603.5622, Y 2.7004, Z -6.3333, A 0.000, B 0.000, C 0.000 }
gfCNCPoint5[5945] = {X 603.6311, Y 2.8108, Z -6.3333, A 0.000, B 0.000, C 0.000 }
gfCNCPoint5[5946] = {X 603.6966, Y 2.9233, Z -6.3333, A 0.000, B 0.000, C 0.000 }
gfCNCPoint5[5947] = {X 607.8227, Y 10.2681, Z -6.3333, A 0.000, B 0.000, C 0.000 }
gfCNCPoint5[5948] = {X 607.8227, Y 10.2681, Z -3.3333, A 0.000, B 0.000, C 0.000 }
gfCNCPoint5[5949] = {X 607.8227, Y 10.2681, Z 11.0000, A 0.000, B 0.000, C 0.000 }
gfCNCPoint5[5950] = {X 607.6966, Y 39.1583, Z 11.0000, A 0.000, B 0.000, C 0.000 }
gfCNCPoint5[5951] = {X 607.6966, Y 39.1583, Z -3.3333, A 0.000, B 0.000, C 0.000 }
gfCNCPoint5[5952] = {X 607.6966, Y 39.1583, Z -6.3333, A 0.000, B 0.000, C 0.000 }
gfCNCPoint5[5953] = {X 603.6966, Y 46.9080, Z -6.3333, A 0.000, B 0.000, C 0.000 }
gfCNCPoint5[5954] = {X 603.6000, Y 47.0846, Z -6.3333, A 0.000, B 0.000, C 0.000 }
gfCNCPoint5[5955] = {X 603.4950, Y 47.2562, Z -6.3333, A 0.000, B 0.000, C 0.000 }
gfCNCPoint5[5956] = {X 602.9785, Y 47.9041, Z -6.3333, A 0.000, B 0.000, C 0.000 }
gfCNCPoint5[5957] = {X 602.3439, Y 48.4368, Z -6.3333, A 0.000, B 0.000, C 0.000 }
gfCNCPoint5[5958] = {X 601.6162, Y 48.8332, Z -6.3333, A 0.000, B 0.000, C 0.000 }
gfCNCPoint5[5959] = {X 600.8245, Y 49.0775, Z -6.3333, A 0.000, B 0.000, C 0.000 }
gfCNCPoint5[5960] = {X 600.0000, Y 49.1600, Z -6.3333, A 0.000, B 0.000, C 0.000 }
gfCNCPoint5[5961] = {X 593.5565, Y 49.1600, Z -6.3333, A 0.000, B 0.000, C 0.000 }
gfCNCPoint5[5962] = {X 592.6308, Y 49.0557, Z -6.3333, A 0.000, B 0.000, C 0.000 }
gfCNCPoint5[5963] = {X 591.7516, Y 48.7480, Z -6.3333, A 0.000, B 0.000, C 0.000 }
gfCNCPoint5[5964] = {X 590.9628, Y 48.2524, Z -6.3333, A 0.000, B 0.000, C 0.000 }
gfCNCPoint5[5965] = {X 590.3041, Y 47.5937, Z -6.3333, A 0.000, B 0.000, C 0.000 }
gfCNCPoint5[5966] = {X 589.8085, Y 46.8050, Z -6.3333, A 0.000, B 0.000, C 0.000 }
gfCNCPoint5[5967] = {X 589.5008, Y 45.9257, Z -6.3333, A 0.000, B 0.000, C 0.000 }
gfCNCPoint5[5968] = {X 589.3965, Y 45.0000, Z -6.3333, A 0.000, B 0.000, C 0.000 }
gfCNCPoint5[5969] = {X 589.3965, Y 44.0653, Z -6.3333, A 0.000, B 0.000, C 0.000 }
gfCNCPoint5[5970] = {X 589.5007, Y 43.1532, Z -6.3333, A 0.000, B 0.000, C 0.000 }
gfCNCPoint5[5971] = {X 589.8006, Y 42.2856, Z -6.3333, A 0.000, B 0.000, C 0.000 }
gfCNCPoint5[5972] = {X 590.2819, Y 41.5039, Z -6.3333, A 0.000, B 0.000, C 0.000 }
gfCNCPoint5[5973] = {X 590.9216, Y 40.8454, Z -6.3333, A 0.000, B 0.000, C 0.000 }
gfCNCPoint5[5974] = {X 590.9223, Y 32.7112, Z -6.3333, A 0.000, B 0.000, C 0.000 }
gfCNCPoint5[5975] = {X 585.2975, Y 46.5912, Z -6.3333, A 0.000, B 0.000, C 0.000 }
gfCNCPoint5[5976] = {X 584.9414, Y 47.2678, Z -6.3333, A 0.000, B 0.000, C 0.000 }
gfCNCPoint5[5977] = {X 584.4675, Y 47.8677, Z -6.3333, A 0.000, B 0.000, C 0.000 }
gfCNCPoint5[5978] = {X 583.8918, Y 48.3708, Z -6.3333, A 0.000, B 0.000, C 0.000 }
gfCNCPoint5[5979] = {X 583.2338, Y 48.7600, Z -6.3333, A 0.000, B 0.000, C 0.000 }
gfCNCPoint5[5980] = {X 582.3250, Y 49.0678, Z -6.3333, A 0.000, B 0.000, C 0.000 }
gfCNCPoint5[5981] = {X 581.3699, Y 49.1592, Z -6.3333, A 0.000, B 0.000, C 0.000 }
gfCNCPoint5[5982] = {X 580.4192, Y 49.0293, Z -6.3333, A 0.000, B 0.000, C 0.000 }
gfCNCPoint5[5983] = {X 579.5236, Y 48.6850, Z -6.3333, A 0.000, B 0.000, C 0.000 }
gfCNCPoint5[5984] = {X 578.7306, Y 48.1448, Z -6.3333, A 0.000, B 0.000, C 0.000 }
gfCNCPoint5[5985] = {X 578.0826, Y 47.4372, Z -6.3333, A 0.000, B 0.000, C 0.000 }
gfCNCPoint5[5986] = {X 577.6138, Y 46.5999, Z -6.3333, A 0.000, B 0.000, C 0.000 }
gfCNCPoint5[5987] = {X 571.8595, Y 32.5291, Z -6.3333, A 0.000, B 0.000, C 0.000 }
gfCNCPoint5[5988] = {X 571.8598, Y 40.8462, Z -6.3333, A 0.000, B 0.000, C 0.000 }
gfCNCPoint5[5989] = {X 571.9199, Y 40.8956, Z -6.3333, A 0.000, B 0.000, C 0.000 }
gfCNCPoint5[5990] = {X 572.5329, Y 41.5415, Z -6.3333, A 0.000, B 0.000, C 0.000 }
gfCNCPoint5[5991] = {X 572.9945, Y 42.3032, Z -6.3333, A 0.000, B 0.000, C 0.000 }
gfCNCPoint5[5992] = {X 573.2833, Y 43.1455, Z -6.3333, A 0.000, B 0.000, C 0.000 }
gfCNCPoint5[5993] = {X 573.3863, Y 44.0301, Z -6.3333, A 0.000, B 0.000, C 0.000 }
gfCNCPoint5[5994] = {X 573.3864, Y 45.0000, Z -6.3333, A 0.000, B 0.000, C 0.000 }
gfCNCPoint5[5995] = {X 573.2821, Y 45.9257, Z -6.3333, A 0.000, B 0.000, C 0.000 }
gfCNCPoint5[5996] = {X 572.9745, Y 46.8050, Z -6.3333, A 0.000, B 0.000, C 0.000 }
gfCNCPoint5[5997] = {X 572.4788, Y 47.5937, Z -6.3333, A 0.000, B 0.000, C 0.000 }
gfCNCPoint5[5998] = {X 571.8201, Y 48.2524, Z -6.3333, A 0.000, B 0.000, C 0.000 }
gfCNCPoint5[5999] = {X 571.0314, Y 48.7480, Z -6.3333, A 0.000, B 0.000, C 0.000 }
gfCNCPoint5[6000] = {X 570.1521, Y 49.0557, Z -6.3333, A 0.000, B 0.000, C 0.000 }
gfCNCPoint5[6001] = {X 569.2264, Y 49.1600, Z -6.3333, A 0.000, B 0.000, C 0.000 }
gfCNCPoint5[6002] = {X 562.4443, Y 49.1600, Z -6.3333, A 0.000, B 0.000, C 0.000 }
gfCNCPoint5[6003] = {X 561.5186, Y 49.0557, Z -6.3333, A 0.000, B 0.000, C 0.000 }
gfCNCPoint5[6004] = {X 560.6393, Y 48.7480, Z -6.3333, A 0.000, B 0.000, C 0.000 }
gfCNCPoint5[6005] = {X 559.8506, Y 48.2524, Z -6.3333, A 0.000, B 0.000, C 0.000 }
gfCNCPoint5[6006] = {X 559.1919, Y 47.5937, Z -6.3333, A 0.000, B 0.000, C 0.000 }
gfCNCPoint5[6007] = {X 558.6963, Y 46.8050, Z -6.3333, A 0.000, B 0.000, C 0.000 }
gfCNCPoint5[6008] = {X 558.3886, Y 45.9257, Z -6.3333, A 0.000, B 0.000, C 0.000 }
gfCNCPoint5[6009] = {X 558.2843, Y 45.0000, Z -6.3333, A 0.000, B 0.000, C 0.000 }
gfCNCPoint5[6010] = {X 558.2843, Y 44.0654, Z -6.3333, A 0.000, B 0.000, C 0.000 }
gfCNCPoint5[6011] = {X 558.3882, Y 43.1529, Z -6.3333, A 0.000, B 0.000, C 0.000 }
gfCNCPoint5[6012] = {X 558.6884, Y 42.2849, Z -6.3333, A 0.000, B 0.000, C 0.000 }
gfCNCPoint5[6013] = {X 559.1704, Y 41.5032, Z -6.3333, A 0.000, B 0.000, C 0.000 }
gfCNCPoint5[6014] = {X 559.8112, Y 40.8452, Z -6.3333, A 0.000, B 0.000, C 0.000 }
gfCNCPoint5[6015] = {X 559.8112, Y 9.1547, Z -6.3333, A 0.000, B 0.000, C 0.000 }
gfCNCPoint5[6016] = {X 559.1739, Y 8.5051, Z -6.3333, A 0.000, B 0.000, C 0.000 }
gfCNCPoint5[6017] = {X 558.6932, Y 7.7326, Z -6.3333, A 0.000, B 0.000, C 0.000 }
gfCNCPoint5[6018] = {X 558.3919, Y 6.8740, Z -6.3333, A 0.000, B 0.000, C 0.000 }
gfCNCPoint5[6019] = {X 558.2845, Y 5.9704, Z -6.3333, A 0.000, B 0.000, C 0.000 }
gfCNCPoint5[6020] = {X 558.2843, Y 5.0000, Z -6.3333, A 0.000, B 0.000, C 0.000 }
gfCNCPoint5[6021] = {X 558.3886, Y 4.0743, Z -6.3333, A 0.000, B 0.000, C 0.000 }
gfCNCPoint5[6022] = {X 558.6963, Y 3.1950, Z -6.3333, A 0.000, B 0.000, C 0.000 }
gfCNCPoint5[6023] = {X 559.1919, Y 2.4063, Z -6.3333, A 0.000, B 0.000, C 0.000 }
gfCNCPoint5[6024] = {X 559.8506, Y 1.7476, Z -6.3333, A 0.000, B 0.000, C 0.000 }
gfCNCPoint5[6025] = {X 560.6393, Y 1.2520, Z -6.3333, A 0.000, B 0.000, C 0.000 }
gfCNCPoint5[6026] = {X 561.5186, Y 0.9443, Z -6.3333, A 0.000, B 0.000, C 0.000 }
gfCNCPoint5[6027] = {X 562.4443, Y 0.8400, Z -6.3333, A 0.000, B 0.000, C 0.000 }
gfCNCPoint5[6028] = {X 570.9376, Y 0.8400, Z -6.3333, A 0.000, B 0.000, C 0.000 }
gfCNCPoint5[6029] = {X 571.8632, Y 0.9443, Z -6.3333, A 0.000, B 0.000, C 0.000 }
gfCNCPoint5[6030] = {X 572.7425, Y 1.2520, Z -6.3333, A 0.000, B 0.000, C 0.000 }
gfCNCPoint5[6031] = {X 573.5313, Y 1.7476, Z -6.3333, A 0.000, B 0.000, C 0.000 }
gfCNCPoint5[6032] = {X 574.1900, Y 2.4063, Z -6.3333, A 0.000, B 0.000, C 0.000 }
gfCNCPoint5[6033] = {X 574.6856, Y 3.1950, Z -6.3333, A 0.000, B 0.000, C 0.000 }
gfCNCPoint5[6034] = {X 574.9933, Y 4.0743, Z -6.3333, A 0.000, B 0.000, C 0.000 }
gfCNCPoint5[6035] = {X 575.0976, Y 5.0000, Z -6.3333, A 0.000, B 0.000, C 0.000 }
gfCNCPoint5[6036] = {X 575.0976, Y 5.9342, Z -6.3333, A 0.000, B 0.000, C 0.000 }
gfCNCPoint5[6037] = {X 575.0212, Y 6.7273, Z -6.3333, A 0.000, B 0.000, C 0.000 }
gfCNCPoint5[6038] = {X 574.7951, Y 7.4913, Z -6.3333, A 0.000, B 0.000, C 0.000 }
gfCNCPoint5[6039] = {X 574.4275, Y 8.1982, Z -6.3333, A 0.000, B 0.000, C 0.000 }
gfCNCPoint5[6040] = {X 581.1907, Y 24.7925, Z -6.3333, A 0.000, B 0.000, C 0.000 }
gfCNCPoint5[6041] = {X 588.0237, Y 8.0809, Z -6.3333, A 0.000, B 0.000, C 0.000 }
gfCNCPoint5[6042] = {X 587.7000, Y 7.4163, Z -6.3333, A 0.000, B 0.000, C 0.000 }
